(* CoDeSys 2.3.9.59 project: wago_880.pro *)
(* Libraries: WagoLibMBX_01.lib 23.7.19 10:23:10, DALI_647_02_v2.3.lib 13.9.26 18:52:45, DALI_02_v2.14.lib 13.9.26 18:52:45, WagoLibReset.lib 2.12.10 14:48:32, DMXStageProfi_01.lib 13.9.26 18:52:45, SysLibFile.lib 2.12.10 14:48:34, Visual.lib 2.12.10 14:48:34, WagoLibEthernet_01.lib 10.7.18 07:47:36, SysLibSockets.lib 10.2.11 09:20:54, mod_com.lib 2.12.10 14:48:32, KNX_Standard.lib 13.9.26 18:52:45, KNX_IP_750_849_01.lib 13.9.26 18:52:45, Ethernet.lib 2.12.10 14:48:32, SysLibGetAddress.lib 2.12.10 14:48:32, WAGOLibKNXDevice.lib 1.4.16 09:47:39, DALI_647_SensorType2_02.lib 13.9.26 18:52:45, DALI_647_SensorType1_02.lib 13.9.26 18:52:45, Standard.lib 2.12.10 14:48:34, SYSLIBCALLBACK.LIB 2.12.10 14:48:32 *)

(* PLC configuration (modules and I/O channels)
K-Bus [K_Bus] node 0, in %IB0 out %QB0
Fieldbus variables [FB_VARS] node 1, in %IB512 out %QB512
*)

(* Global variable list: Variables_Globales *)
VAR_GLOBAL CONSTANT
	MaxDaliSensors: BYTE := 128;
END_VAR
VAR_GLOBAL
	ConfigDone: BOOL := FALSE; (* Do the config only one time *)
	info : ARRAY[0..63] OF MODULE_INFO; (* I/O Module infos *)

	LedMode: BYTE := 0;

	(* modules infos *)
	nb_module: BYTE;
	nb_module_in: BYTE;
	nb_module_out: BYTE;
	nb_module_analog_in: BYTE;
	nb_module_analog_out: BYTE;
	start_addr_in: WORD;
	start_addr_out: WORD;
	nb_input_digital: WORD;
	nb_output_digital: WORD;

	(* All inputs events *)
	event: ARRAY[0..512] OF INTER_EVENT; (* See Rules mapping below *)
	lights: ARRAY[0..63] OF BYTE;	(* MAX of 256/8 = 32 digital output modules as lights *)
									(* We store only the boolean state of each light *)
	volets: ARRAY[0..512] OF VOLET; (* MAX of 256/8 = 32 digital output modules as volets *)

	HEARTBEAT: BOOL := FALSE;

	OutArrState: ARRAY[0..512] OF BYTE;	(* state of outputs *)

	impulse_time: TIME := T#300ms;

	(* DALI *)
	DALIJoblist: FbDALI_Joblist;

	Dali_switch: DaliSwitch;
	DALIDimmValue: DaliDimValue;
	DALIShowShortAdr: FbDALI_ShowShortAdr;

	(* DALI 647 module *)
	DaliSendValue647: ARRAY[1..64] OF FbDaliSendDimmValue;
	DaliSendValueGrp647: ARRAY[1..16] OF FbDaliSendDimmValue;
	DaliValue647: ARRAY[1..64] OF BYTE;
	DaliValueGrp647: ARRAY[1..16] OF BYTE;

	daliSensors: ARRAY [1..MaxDaliSensors] OF typDaliSensorData;
	DaliSensorT1: ARRAY[1..MaxDaliSensors] OF FbMultiSensorType1;
	DaliButtonT1: ARRAY[1..MaxDaliSensors] OF FbPushbuttonSensorType1;
	DaliSensorT2: ARRAY[1..MaxDaliSensors] OF FbMultiSensorType2;
	DaliButtonT2: ARRAY[1..MaxDaliSensors] OF FbPushbuttonSensorType2;

	(* DALI sensors input mapping *)
	DaliSensorsInputs: ARRAY[0..768] OF BOOL;

	(*
		Modbus addresses mapping:
			- [4096..4352] : Standard digital outputs
			- [6144..6248] : KNX inputs/outputs
			- [6656..7424] : Dali Master Sensors Digital (max 768 addresses available)
			- [256..272] : Dali Master Sensors Analog values (16 addresses for lightlevels in WORD)
	*)

	netOutStandard AT %IB512: ARRAY[0..31] OF BYTE;

	netDaliSensor AT %QB832: ARRAY[0..31] OF BYTE; (* addresses for digital values *)
	netDaliLevels AT %QW256: ARRAY[0..15] OF WORD; (* addresses for light levels *)

	write_word: WRITE_OUTPUT_WORD;
	read_word: READ_INPUT_WORD;
	write_bit: WRITE_OUTPUT_BIT;
	read_bit: READ_INPUT_BIT;

END_VAR
VAR_GLOBAL RETAIN
	(* Rules mapping:
		- [0..256] : standard digital inputs
		- [257..357]: knx digital inputs
	*)
	output_type: ARRAY[0..512] OF OUTPUT_TYPE; (* The type of each output *)
	output_addr: ARRAY[0..512] OF OUTPUT_ADDR; (* The addresses for each type *)

   	volets_position: ARRAY[0..100] OF DWORD;

	(* DMX Values *)
	abDMX_Values: ARRAY [1..255] OF BYTE;
END_VAR

(* Data type *)
TYPE enumDaliSensor :
(
	NoSensor := 0, (* default type is no sensor *)
	MultiSensorType1,
	PushbuttonSensorType1,
	MultiSensorType2,
	PushbuttonSensorType2,
	DaliEcg,
	DaliGroup
);
END_TYPE

(* Data type *)
TYPE OUTPUT_ADDR :
STRUCT

	(* the first ouput address, only needed *)
	ADDR1: BYTE;
	(* the second address used only for the VOLET function bloc *)
	ADDR2: BYTE;

	(* If SameAs <> -1, then a input is wired the same as the specified ID *)
	SameAs: INT := -1;

END_STRUCT
END_TYPE

(* Data type *)
(* Enumerate all type of output.
	NONE: Do nothing.
	TELERUPTEUR: Simulate a telerupteur.
	DIRECT: The input is directly "wired" to the output.
	VOLET: Simulate a volet with one button and 2 output (up and down).
	TELERUPTEUR_DALI: Controls a DALI lamp
	TELERUPTEUR_DALI_GROUP: Controls a DALI group
	KNX_OUTPUT: Simulate a telerupteur with a KNX bool output
*)

TYPE OUTPUT_TYPE : (NONE,
					TELERUPTEUR, DIRECT,
					VOLET, VOLET_IMPULSE,
					TELERUPTEUR_DALI,
					TELERUPTEUR_DALI_GROUP,
					TELERUPTEUR_KNX_OUTPUT,
					DIRECT_KNX_OUTPUT);
END_TYPE

(* Data type *)
TYPE typDaliSensorData :
STRUCT

	SensorType: enumDaliSensor;

	(* MultiSensorType1 *)
	AddrPresence: BYTE;
	AddrLightLevel: BYTE;
	offDelay: TIME;

	(* MultiSensorType2 *)
	AddrRemote: BYTE;

	(* PushbuttonSensorType1 *)
	AddrButton1: BYTE;
	AddrButton2: BYTE;
	AddrButton3: BYTE;
	AddrButton4: BYTE;

	(* PushbuttonSensorType2 *)
	AddrButtons: BYTE;

	(* Dali devices *)
	Address: BYTE;

END_STRUCT
END_TYPE

(* Data type *)
TYPE typEthernet_BUFFER :
	STRUCT
		Index		:	INT;
		Data		:	ARRAY[1..1500] OF BYTE;
	END_STRUCT
END_TYPE

(* Data type *)
(* Enumerate all type of output.
	NONE: Do nothing.
	TELERUPTEUR: Simulate a telerupteur.
	DIRECT: The input is directly "wired" to the output.
	VOLET: Simulate a volet with one button and 2 output (up and down).
*)

TYPE VOLET_MODE : (VOLET_STOP, VOLET_UP, VOLET_DOWN, IMP_UP, IMP_DOWN, IMP_STOP);
END_TYPE

(* POU PLC_PRG, ST *)
PROGRAM PLC_PRG
VAR
	i: INT;
	j: INT;
	start: BYTE;
	init_dali: BOOL := FALSE;
	valw: WORD;

	led: LedUsr;

END_VAR
(* Main PRG *)
Config_File_XML();

(*DaliReadCsvFile(xStart := TRUE);*)

led(Mode := LedMode);

(* Start the config program *)
Config;

IF (Config.CONFIG_DALI = TRUE) THEN
	(* Call DALI jobs to send commands on the DALI bus *)
	DALIJoblist();
	DALI_Config();
END_IF

(* Read inputs and send their status on the network if they changed *)
SendInput;

(* Read a command from UDP *)
UDPServer;

IF (HEARTBEAT = FALSE) THEN
 	ManageOutput;
END_IF

(* Run the DALI FB for 647 module *)
IF Config.CONFIG_DALI_647 = TRUE THEN
	DaliPrg647;
END_IF

IF (HEARTBEAT = FALSE) THEN

	j := start_addr_out / 8;
	FOR i := start_addr_out / 16 TO 255 DO
		valw := OutArrState[j + 1];
		write_word(WORD_ADDRESS := i, VALUE := SHL(valw, 8) + OutArrState[j]);
		j := j + 2;
	END_FOR
ELSE

	j := 0;
	FOR i := 0 TO 14 DO
		valw := netOutStandard[j + 1];
		write_word(WORD_ADDRESS := i + start_addr_out / 16, VALUE := SHL(valw, 8) + netOutStandard[j]);
		j := j + 2;
		OutArrState[j] := netOutStandard[j];
		OutArrState[j + 1] := netOutStandard[j + 1];
	END_FOR

END_IF
END_PROGRAM

(* POU LedUsr, ST *)
FUNCTION_BLOCK LedUsr
VAR_INPUT
	Mode: BYTE;

END_VAR
VAR_OUTPUT
END_VAR
VAR
	Sequence: ARRAY [0..4] OF FLASHING_SEQUENCE;
	ptrFS: POINTER TO FLASHING_SEQUENCE;

	i: BYTE := 0;
END_VAR
CASE Mode OF
	0 : i := 0;
	1 : i := 11; (* Mode Wago *)
	2 : i := 12; (* Mode PC *)
	3 : i := 13; (* Error *)
END_CASE

LedMode := 255;

CASE i OF
	0 : (* Init *)
		Sequence[0].Colour := ORANGE;
		Sequence[0].Frequency := 10;
		Sequence[0].Relation := 128;
		Sequence[0].Duration := t#0s;

		Sequence[1].Colour := ORANGE;
		Sequence[1].Frequency := 0;
		Sequence[1].Relation := 128;
		Sequence[1].Duration := t#0s;

		Sequence[2].Colour := GREEN;
		Sequence[2].Frequency := 0;
		Sequence[2].Relation := 128;
		Sequence[2].Duration := t#0s;

		Sequence[3].Colour := RED;
		Sequence[3].Frequency := 0;
		Sequence[3].Relation := 128;
		Sequence[3].Duration := t#0s;

		Sequence[4].Colour := ORANGE;
		Sequence[4].Frequency := 0;
		Sequence[4].Relation := 0;
		Sequence[4].Duration := t#0s;

		ptrFS := ADR(Sequence);
		SET_FLASHING_SEQUENCE(TRUE, ADR(ptrFS));

		i := 10;

	10: (* Start *)
		SET_FLASHING_SEQUENCE_INDEX(TRUE, TRUE, 0);
		START_FLASHING_SEQUENCE(TRUE);

		i := 255;

	11: (* Led Mode wago *)
		SET_FLASHING_SEQUENCE_INDEX(TRUE, TRUE, 1);

		i := 255;

	12: (* Led Mode PC *)
		SET_FLASHING_SEQUENCE_INDEX(TRUE, TRUE, 2);

		i := 255;

	13: (* Led Error *)
		SET_FLASHING_SEQUENCE_INDEX(TRUE, TRUE, 3);

		i := 255;

END_CASE
END_FUNCTION_BLOCK

(* POU Config_File_XML, ST *)
PROGRAM Config_File_XML
VAR RETAIN
	wModuleCount : WORD;
END_VAR
VAR CONSTANT
	STRING_1: STRING := '<?xml version="1.0" encoding="ISO-8859-1"?>$r$n';
	STRING_2: STRING := '<?xml-stylesheet type="text/xsl" href="/webserv/cplcfg/EA-config.xsl" ?>$R$n';
	STRING_3: STRING := '<WAGO>$R$n';
	STRING_4: STRING := '<Module ARTIKELNR="" MAP="PLC" LOC="ALL"></Module>$R$n';
	STRING_5: STRING := '</WAGO>$r$n';
END_VAR
VAR
	info : ARRAY[0..63] OF MODULE_INFO;
	access: MODULE_INFO_ACCESS;
	i: INT := 0;
	Status: BYTE := 0;
	DetectedModules: INT;
	FileHandle: DWORD;
	dwWrite: DWORD;
	NumberOfEntries: BYTE := 0;
	FileIsClosed: BOOL;
END_VAR
CASE Status OF
	0 :	ADD_PI_INFORMATION(EN:=TRUE, pAccess:=ADR(access), pInfo:=ADR(info));
		i:=0;
		WHILE info[i].physicalPos<>0
			DO
			i:=i+1;
		END_WHILE
		DetectedModules := i;
		Status := Status +1;
	1 :	IF DetectedModules = wModuleCount
			THEN
			Status := 255; (* Done *)
		ELSE
			Status := 10;
		END_IF
	10:	FileHandle:=SysFileOpen(FileName:='\etc\EA-config.xml', Mode:='w');
		IF FileHandle <> 0 THEN
			Status := Status+1;
		END_IF
	11:	dwWrite:=SysFileWrite(File:=FileHandle, Buffer:=ADR(STRING_1), Size:=LEN(STRING_1));
		IF dwWrite=LEN(STRING_1) THEN
			Status := Status+1;
		END_IF
	12:	dwWrite:=SysFileWrite(File:=FileHandle, Buffer:=ADR(STRING_2), Size:=LEN(STRING_2));
		IF dwWrite=LEN(STRING_2) THEN
			Status := Status+1;
		END_IF
	13:	dwWrite:=SysFileWrite(File:=FileHandle, Buffer:=ADR(STRING_3), Size:=LEN(STRING_3));
		IF dwWrite=LEN(STRING_3) THEN
			Status := Status+1;
		END_IF
	14:	dwWrite:=SysFileWrite(File:=FileHandle, Buffer:=ADR(STRING_4), Size:=LEN(STRING_4));
		IF dwWrite=LEN(STRING_4) THEN
			Status := Status+1;
			NumberOfEntries := NumberOfEntries+1;
		END_IF
	15: IF NumberOfEntries < DetectedModules
			THEN
			Status := Status -1;
		ELSE
			Status := Status +1;
		END_IF
	16:	dwWrite:=SysFileWrite(File:=FileHandle, Buffer:=ADR(STRING_5), Size:=LEN(STRING_5));
		IF dwWrite=LEN(STRING_5) THEN
			Status := Status+1;
		END_IF
	17:	FileIsClosed := SysFileClose(File:= FileHandle);
		IF FileIsClosed
			THEN
			Status := 20;
		END_IF
	20:	wModuleCount := DetectedModules;
		FirmwareReset(EN := TRUE);
END_CASE
END_PROGRAM

(* POU Config, ST *)
PROGRAM Config
VAR
	access : MODULE_INFO_ACCESS;
	cpt: BYTE;
	ethernet_config : ETHERNET_SET_VARIABLES;
	CONFIG_DALI: BOOL := FALSE;
	CONFIG_DALI_647: BOOL := FALSE;
	first_in: BOOL := FALSE;
	first_out: BOOL := FALSE;
	AddrDali647In: INT;
	AddrDali647Out: INT;
END_VAR
VAR_INPUT RETAIN
	SERVER_IP: DWORD;
	DALI_MODE: BYTE;
END_VAR
VAR CONSTANT
	CALAOS_VERSION_H: WORD := 3;
	CALAOS_VERSION_L: WORD := 0;
	DALI: BYTE := 1;
	DSI: BYTE := 2;
END_VAR
(* Do all the config job *)

IF (ConfigDone = FALSE) THEN

(* Get the module I/O Config *)
access.physicalPosTo := 0;
access.moduleType := 0;
ADD_PI_INFORMATION( 1, ADR(access), ADR(info[0]) );

FOR cpt := 0 TO 63 DO
	IF (info[cpt].moduleType = 0 AND info[cpt].physicalPos = 0) THEN
		cpt := 63; (* the end *)
	ELSE
		IF (info[cpt].moduleType = 641) THEN
			(* This is a DALI 641 module *)
			CONFIG_DALI := TRUE;
		END_IF

		IF (info[cpt].moduleType = 647) THEN
			(* This is a DALI 753-647 module (multi master) *)
			CONFIG_DALI_647 := TRUE;
		END_IF

		nb_module := nb_module + 1;
		IF ((info[cpt].desc.sizePAE > 8) AND (info[cpt].desc.channels > 0)) THEN
			nb_module_analog_in := nb_module_analog_in + 1;
(*			start_addr_in := start_addr_in + info[cpt].desc.sizePAE; *)
			IF CONFIG_DALI_647 = FALSE THEN
				AddrDali647In := AddrDali647In + (info[cpt].desc.sizePAE / 8);
			END_IF
		END_IF
		IF ((info[cpt].desc.sizePAA > 8) AND (info[cpt].desc.channels > 0)) THEN
			nb_module_analog_out := nb_module_analog_out + 1;
(*			start_addr_out := start_addr_out + info[cpt].desc.sizePAA; *)
			IF CONFIG_DALI_647 = FALSE THEN
				AddrDali647Out := AddrDali647Out + (info[cpt].desc.sizePAA / 8);
			END_IF
		END_IF
		IF ((info[cpt].desc.sizePAE <= 16) AND (info[cpt].desc.sizePAE > 0) AND (info[cpt].desc.channels = 0)) THEN
			nb_module_in := nb_module_in + 1;
			nb_input_digital := nb_input_digital + info[cpt].desc.sizePAE;

			IF (first_in = FALSE) THEN
				first_in := TRUE;
				start_addr_in := info[cpt].desc.posPAE;
			END_IF
		END_IF
		IF ((info[cpt].desc.sizePAA <= 16) AND (info[cpt].desc.sizePAA > 0) AND (info[cpt].desc.channels = 0)) THEN
			nb_module_out := nb_module_out + 1;
			nb_output_digital := nb_output_digital + info[cpt].desc.sizePAA;

			IF (first_out = FALSE) THEN
				first_out := TRUE;
				start_addr_out := info[cpt].desc.posPAA;
			END_IF
		END_IF

	END_IF
END_FOR

(* Start the heartbeat timer *)
(*HEARTBEAT_TIMER(IN:=FALSE, PT:=T#30s);*)
(*HEARTBEAT_TIMER(IN:=TRUE, PT:=T#30s);*)

(* Config du timout des sockets *)
ethernet_config(EN:=TRUE, BootpRequest:=0, ConnectionWdTime:=65535);

ConfigDone := TRUE;

END_IF
END_PROGRAM

(* POU SendInput, ST *)
PROGRAM SendInput
VAR
	cpt: INT;

	eth: Ethernet_Client;
	wBuffer: POINTER TO BYTE;
	command: STRING(255);
	start_send: BOOL := FALSE;
	ReceiveData: typEthernet_buffer;
	Write: ETHERNET_WRITE_PT;
	socket:	WORD;
END_VAR
(* Get all inputs *)

(* Get the address of the first digital input *)
FOR cpt := 0 TO UINT_TO_BYTE(nb_input_digital) - 1 DO
	event[cpt](IN := GetInput(cpt + start_addr_in));

	(* Send inputs to network *)
	IF (event[cpt].ON = TRUE) THEN
		command := 'WAGO INT ';
		command := CONCAT(command,  INT_TO_STRING(cpt));
		command := CONCAT(command,  ' 1');

		Write(EN := 0, SOCKET := 0, LEN_IN := 0, DST_IP:=0, DST_PORT:=0, DATA_PT := wBuffer);
		Write(EN := 1, SOCKET := socket, LEN_IN := LEN(command), DST_IP := Config.SERVER_IP, DST_PORT := 4646, DATA_PT := wBuffer);
	END_IF
	IF (event[cpt].OFF = TRUE) THEN
		command := 'WAGO INT ';
		command := CONCAT(command,  INT_TO_STRING(cpt));
		command := CONCAT(command,  ' 0');

		Write(EN := 0, SOCKET := 0, LEN_IN := 0, DST_IP:=0, DST_PORT:=0, DATA_PT := wBuffer);
		Write(EN := 1, SOCKET := socket, LEN_IN := LEN(command), DST_IP := Config.SERVER_IP, DST_PORT := 4646, DATA_PT := wBuffer);
	END_IF
END_FOR

wBuffer := ADR(command);

eth(xOPEN_CLIENT := TRUE, wIP := Config.SERVER_IP, wPort := 4646,
	xTCP_PROTOCOL := FALSE, iBYTES_TO_SEND := LEN(command) + 1,
	ptSEND_BUFFER := wBuffer, xSTART_SEND := start_send,
	utRECEIVE_BUFFER := ReceiveData);

socket := eth.MyEthernetOpen.SOCKET;
END_PROGRAM

(* POU Ethernet_Client, ST *)
FUNCTION_BLOCK Ethernet_Client
(************************************************************)
(* ETHERNET_CLIENT		                             			*)
(* Ver. 1.0                                      			          			*)
(* Date    :  10.02.2003					          			*)
(* Author :  Volker Begemann                                       		*)
(************************************************************)
VAR_INPUT
	xOPEN_CLIENT			:	BOOL;			(* Set TRUE to enable function block			*)
	wIP						:	DWORD;		(* IP Address of server						*)
	wPORT					:	WORD;		(* Port number								*)
	xTCP_PROTOCOL		:	BOOL;			(* TRUE => TCP; FALSE => UDP				*)
	iBYTES_TO_SEND		:	INT;			(* Number of bytes to transmit				*)
	ptSEND_BUFFER			:	POINTER TO ARRAY[1..1500] OF BYTE;	(* Transmit Buffer	*)
END_VAR
VAR_IN_OUT
	xSTART_SEND			:	BOOL;			(* Set TRUE to initiate data transmittal, will be	*)
													(* reset FALSE when transmittal is completed 	*)
	utRECEIVE_BUFFER		:	typEthernet_BUFFER;	(* Receive Buffer *)
END_VAR
VAR_OUTPUT
	utERROR					:	ETH_ERROR;	(* See ETH_ERROR datatype in ETHERNET.LIB	*)
													(* for error codes and definitions						*)
	xCLIENT_OPEN			:	BOOL;			(* TRUE if socket connection made					*)
	wSOCKET					:	WORD;		(* Socket connection number							*)
END_VAR
VAR
	MyEthernetOpen				: ETHERNET_CLIENT_OPEN;
	MyEthernetClose				: ETHERNET_CLIENT_CLOSE;
	MyEthernetWrite				: ETHERNET_WRITE;
	MyEthernetRead				: ETHERNET_READ;
	EthernetBuffer					: ARRAY[1..1500] OF BYTE;
	Status							: WORD:=0;
	i								: INT;
	GetConfig						: ETHERNET_GET_NETWORK_CONFIG;
	Protocol						: WORD;
	ProtocolType					: WORD;
	CloseState						:INT;
END_VAR
IF xOpen_Client THEN

	CASE Status OF
		0:(*Initialize functionblocks*)
			GetConfig(EN:=FALSE );
			GetConfig(EN:=TRUE );
			status:=1;
			utERROR:=0;
			wSocket:=0;
			closeState:=0;
			xCLIENT_OPEN:=FALSE;

			IF xTCP_PROTOCOL THEN
				Protocol		:= IPPROTO_TCP; (*TCP*)
				ProtocolType	:= SOCK_STREAM;
			ELSE
				Protocol		:= IPPROTO_UDP;(*UDP*)
				ProtocolType	:= SOCK_DGRAM;
			END_IF

		1:(*check ethernet stack*)
			GetConfig(EN:=TRUE );
			IF GetConfig.ENO THEN
				IF GetConfig.IP_ADR<>0 THEN
					status:=4;(*stack initialized*)
				ELSE
					status:=0;(*try again*)
				END_IF
			END_IF

	
		4:(*open connection*)
			MyEthernetRead(	EN:= 0, SOCKET:=0 ,  DATA:=EthernetBuffer );
			MyEthernetClose(EN:= 0);
			MyEthernetOpen(EN:=0);

			MyEthernetOpen(EN:=1 , TYP:=ProtocolType	 , PROTO:=Protocol , IP_ADR:= wIP, PORT:=wPort );

			status:=5;

		5:(*wait for server response according to client  request to open the connection*)
			MyEthernetOpen(EN:=1, TYP:=ProtocolType, PROTO:=Protocol, IP_ADR:= wIP, PORT:=wPort );
			IF  MyEthernetOpen.ENO = 1 THEN
				IF MyEthernetOpen.ERROR = 0 THEN
					Status  := 10; (*socket available*)
					xCLIENT_OPEN:=TRUE;
					wSOCKET	:=MyEthernetOpen.socket;
				ELSE
					Status := 0; (*no socket available, try it again *)
				END_IF;
				utERROR:=MyEthernetOpen.ERROR;
			END_IF


		10:(* Monitor ethernet port for new data *)

	 		MyEthernetRead(	EN:= 1, SOCKET:=MyEthernetOpen.SOCKET ,  DATA:=EthernetBuffer );
			MyEthernetRead(	EN:= 0, SOCKET:=0 ,  DATA:=EthernetBuffer );

			utERROR:=MyEthernetREAD.ERROR;
			IF(MyEthernetRead.ERROR<>0) THEN  (* Error reading the socket, close it *)
				Status:=40;
			ELSIF (MyEthernetRead.LEN_OUT <>0) THEN  (* Process the data received via the ethernet port *)
				Status:=20;
				ELSIF (iBytes_TO_SEND > 0 AND xSTART_SEND) THEN  (* Process the data put in the send_buffer *)
				status:=30;
				MyEthernetWrite(	EN:= 0 , DATA:=EthernetBuffer );
			END_IF

		20:	(* Copy the data received via the ethernet port to the receive buffer*)

			FOR i := 1 TO MyEthernetRead.LEN_OUT DO
				utReceive_buffer.index :=(utReceive_buffer.index MOD 1500)+1;
				utReceive_buffer.data[utReceive_buffer.index] := EthernetBuffer[i];
			END_FOR
			Status:=10;

		30: (* Process the data in the send buffer *)

			EthernetBuffer :=ptSEND_BUFFER^;
			MyEthernetWrite(	EN:= 1,SOCKET:= MyEthernetOpen.SOCKET,
								LEN_IN:=iBYTES_TO_SEND,DATA:=EthernetBuffer );

			IF MyEthernetWrite.eno THEN
				IF(MyEthernetWrite.ERROR <>0) THEN
					Status:=40;(* Error writing to the socket, close it *)
				ELSE
					Status:=10; (* Comms complete, read more data *)
				END_IF;
				xSTART_SEND:=FALSE;
				utERROR:=MyEthernetWrite.ERROR;
			END_IF

		40:	(* Close the client *)

			MyEthernetClose(EN:= 1, SOCKET:= MyEthernetOpen.SOCKET);
			IF MyEthernetClose.eno THEN
				MyEthernetClose(EN:= 0);
				xCLIENT_OPEN:=FALSE;
				Status := 0; (* Try to open the server again *)
			END_IF
	
	END_CASE;
ELSE
	CASE CloseState OF
	0:
		MyEthernetClose(EN:= 0);
		MyEthernetClose(EN:= 1, SOCKET:= MyEthernetOpen.SOCKET);
		CloseState:=1;
	1:
		MyEthernetClose(EN:= 1, SOCKET:= MyEthernetOpen.SOCKET);
		IF MyEthernetClose.eno THEN
			MyEthernetClose(EN:= 0);
			CloseState:=2;
		END_IF
	2:
		Status := 0;
		utERROR:=0;
		xCLIENT_OPEN:=FALSE;
	END_CASE
END_IF
END_FUNCTION_BLOCK

(* POU GetInput, ST *)
FUNCTION GetInput : BOOL
VAR_INPUT
	bit_offset: UINT;
END_VAR
VAR
END_VAR
VAR CONSTANT
	byBitArr: ARRAY[0..7] OF BYTE := 16#01,16#02,16#04,16#08,16#10,16#20,16#40,16#80;
END_VAR
(* get the byte AND  select the bit *)

read_bit(WORD_ADDRESS := bit_offset / 16, BIT_ADDRESS := bit_offset MOD 16);

GetInput := read_bit.VALUE;
END_FUNCTION

(* POU UDPServer, ST *)
PROGRAM UDPServer
VAR
	server: EthernetServer_FB;

	rBuffer, wBuffer: POINTER TO BYTE;
	buffer: ARRAY[1 .. 1500] OF BYTE;
	cmd: STRING(255);
	start_send: BOOL := FALSE;
	i: WORD;
	dali_group: BOOL;

	HEARTBEAT_TIMER: TON;

	p1: DINT;
	p2: DINT;
	p3: DINT;
	p4: DINT;
	p5: DINT;
	p6: DINT;
	p7: DINT;
	p8: DINT;
	ip1, ip2, ip3, ip4: DWORD;
	DaliSend: BOOL := FALSE;

	(* Used by dali config for answer
	   0 = no action
	   1 = Search all active address
	   2 = Read groups for short adress
	   3 = Switch on/off all lamps
	  98 = Addresing query
	  99 = Addressing in progress
	*)
	DaliSendAction: BYTE := 0;

	(* Dali config FB *)
	DALIShowShortAdr: FbDALI_ShowShortAdr;
	DALIConfigDevice: FbDALI_ConfigDevice;
	DALIConfigShortAddress: FbDALI_ConfigShortAddress;
	DALIMaster: FbDALI_Master;
	DALIMasterAdv: FbDALI_Master_Adv;

	extendedAddr: BOOL;
	newAddressing: BOOL;
	resetAddr: BOOL;
	replaceAddr: BOOL;
	delAddressing: BOOL;
	oldAddr, newAddr, delAddr: BYTE;
	dali_master: BOOL;
	group_address: BYTE;
	groups_cmd_1_8: BYTE;
	addr_1_16: WORD;
	addr_17_32: WORD;

	dmx_read_addr: BYTE;

	daliShortAddr: BYTE;

END_VAR
(* Here we start an UDP server for other network functions *)

HEARTBEAT_TIMER(IN:=TRUE, PT:=T#30s);

rBuffer := ADR(buffer);
wBuffer := ADR(cmd);

(* cmd := CONCAT(cmd, ASCIIBYTE_TO_STRING(0)); *)

server.tTIMEOUT	:= t#60s;
server.xTCP_PROTOCOL := FALSE;
server.wPORT := 4646;
server.iBYTES_TO_SEND := LEN(cmd) + 1;
server(xOPEN_SERVER := TRUE, xSTART_SEND := start_send, ptSEND_BUFFER := wBuffer, ptRECV_BUFFER := rBuffer);

IF server.bDataReceived THEN

	cmd := '';
	FOR i := 1 TO server.iBYTES_RECEIVED DO
		cmd := CONCAT(cmd, ASCIIBYTE_TO_STRING(buffer[i]));
	END_FOR

	IF (STRING_COMPARE(cmd, 'WAGO_HEARTBEAT') = TRUE) THEN
		HEARTBEAT_TIMER(IN:=FALSE, PT:=T#30s);
		HEARTBEAT_TIMER(IN:=TRUE, PT:=T#30s);

		LedMode := 2;
	END_IF

	IF (Strncmp(cmd, 'WAGO_SET_OUTTYPE ', 17) = TRUE) THEN
		p1 := GET_PARAM_DINT(cmd, 1);
		p2 := GET_PARAM_DINT(cmd, 2);
		CASE p2 OF
		0: output_type[p1] := NONE;
		1: output_type[p1] := TELERUPTEUR;
		2: output_type[p1] := DIRECT;
		3: output_type[p1] := VOLET;
		4: output_type[p1] := VOLET_IMPULSE;
		5: output_type[p1] := TELERUPTEUR_DALI;
		6: output_type[p1] := TELERUPTEUR_DALI_GROUP;
		7: output_type[p1] := TELERUPTEUR_KNX_OUTPUT;
		8: output_type[p1] := DIRECT_KNX_OUTPUT;
		END_CASE
	END_IF

	IF (Strncmp(cmd, 'WAGO_SET_OUTADDR ', 17) = TRUE) THEN
		p1 := GET_PARAM_DINT(cmd, 1);
		p2 := GET_PARAM_DINT(cmd, 2);
		p3 := GET_PARAM_DINT(cmd, 3);
		p4 := GET_PARAM_DINT(cmd, 4);
		output_addr[p1].ADDR1 := DINT_TO_BYTE(p2);
		output_addr[p1].ADDR2 := DINT_TO_BYTE(p3);
		output_addr[p1].SameAs := DINT_TO_INT(p4);
	END_IF

	IF (Strncmp(cmd, 'WAGO_GET_OUTTYPE ', 17) = TRUE) THEN
		p1 := GET_PARAM_DINT(cmd, 1);
		cmd := 'WAGO_OUTTYPE ';
		cmd := CONCAT(cmd, ITOA(DINT_TO_INT(p1)));
		cmd := CONCAT(cmd, ' ');
		CASE output_type[p1] OF
		NONE: cmd := CONCAT(cmd, ITOA(0));;
		TELERUPTEUR: cmd := CONCAT(cmd, ITOA(1));;
		DIRECT: cmd := CONCAT(cmd, ITOA(2));;
		VOLET: cmd := CONCAT(cmd, ITOA(3));;
		VOLET_IMPULSE: cmd := CONCAT(cmd, ITOA(4));;
		TELERUPTEUR_DALI: cmd := CONCAT(cmd, ITOA(5));;
		TELERUPTEUR_DALI_GROUP: cmd := CONCAT(cmd, ITOA(6));;
		TELERUPTEUR_KNX_OUTPUT: cmd := CONCAT(cmd, ITOA(7));;
		DIRECT_KNX_OUTPUT: cmd := CONCAT(cmd, ITOA(8));;
		END_CASE
		start_send := TRUE;
	END_IF

	IF (Strncmp(cmd, 'WAGO_GET_OUTADDR ', 17) = TRUE) THEN
		p1 := GET_PARAM_DINT(cmd, 1);
		cmd := 'WAGO_OUTADDR ';
		cmd := CONCAT(cmd, ITOA(DINT_TO_INT(p1)));
		cmd := CONCAT(cmd, ' ');
		cmd := CONCAT(cmd, ITOA(output_addr[p1].ADDR1));
		cmd := CONCAT(cmd, ' ');
		cmd := CONCAT(cmd, ITOA(output_addr[p1].ADDR2));
		cmd := CONCAT(cmd, ' ');
		cmd := CONCAT(cmd, ITOA(output_addr[p1].SameAs));
		start_send := TRUE;
	END_IF

	IF (STRING_COMPARE(cmd, 'WAGO_GET_INFO') = TRUE) THEN
		cmd := 'WAGO_INFO ';
		cmd := CONCAT(cmd, ITOA(nb_module));
		cmd := CONCAT(cmd, ' ');
		cmd := CONCAT(cmd, ITOA(nb_module_in));
		cmd := CONCAT(cmd, ' ');
		cmd := CONCAT(cmd, ITOA(WORD_TO_INT(nb_module_out)));
		cmd := CONCAT(cmd, ' ');
		cmd := CONCAT(cmd, ITOA(WORD_TO_INT(nb_input_digital)));
		cmd := CONCAT(cmd, ' ');
		cmd := CONCAT(cmd, ITOA(WORD_TO_INT(nb_output_digital)));
		cmd := CONCAT(cmd, ' ');
		cmd := CONCAT(cmd, ITOA(nb_module_analog_in));
		cmd := CONCAT(cmd, ' ');
		cmd := CONCAT(cmd, ITOA(nb_module_analog_out));
		start_send := TRUE;
	END_IF

	IF (Strncmp(cmd, 'WAGO_GET_INFO_MODULE ', 21) = TRUE) THEN
		p1 := GET_PARAM_DINT(cmd, 1);
		cmd := 'WAGO_MODULE ';
		cmd := CONCAT(cmd, ITOA(DINT_TO_INT(p1)));
		cmd := CONCAT(cmd, ' ');
		cmd := CONCAT(cmd, ITOA(WORD_TO_INT(info[p1].moduleType)));
		cmd := CONCAT(cmd, ' ');
		cmd := CONCAT(cmd, ITOA(info[p1].physicalPos));
		cmd := CONCAT(cmd, ' ');
		cmd := CONCAT(cmd, ITOA(info[p1].desc.sizePAE));
		cmd := CONCAT(cmd, ' ');
		cmd := CONCAT(cmd, ITOA(info[p1].desc.sizePAA));
		start_send := TRUE;
	END_IF

	IF (Strncmp(cmd, 'WAGO_SET_SERVER_IP ', 19) = TRUE) THEN
		cmd := DELETE(cmd, 19, 1);
		(* deletes the dot  *)
		cmd := REPLACE(cmd, ' ', 1, FIND(cmd, '.'));
		cmd := REPLACE(cmd, ' ', 1, FIND(cmd, '.'));
		cmd := REPLACE(cmd, ' ', 1, FIND(cmd, '.'));
		ip1 := GET_PARAM_DINT(cmd, 0);
		ip2 := GET_PARAM_DINT(cmd, 1);
		ip3 := GET_PARAM_DINT(cmd, 2);
		ip4 := GET_PARAM_DINT(cmd, 3);
		Config.SERVER_IP := SHL(ip1, 24) OR SHL(ip2, 16) OR SHL(ip3, 8) OR ip4;
	END_IF


	IF (Strncmp(cmd, 'WAGO_SET_DMX_IP ', 16) = TRUE) THEN
		cmd := DELETE(cmd, 16, 1);
		DMX.IPaddress := cmd;
	END_IF

	IF (Strncmp(cmd, 'WAGO_SET_OUTPUT ', 16) = TRUE) THEN
		p1 := GET_PARAM_DINT(cmd, 1);
		p2 := GET_PARAM_DINT(cmd, 2);

		p1 := start_addr_out + p1;

		IF (p2 = 1) THEN
			SetOutput(DINT_TO_UINT(p1), TRUE);
		ELSE
			SetOutput(DINT_TO_UINT(p1), FALSE);
		END_IF
	END_IF

	IF (Strncmp(cmd, 'WAGO_GET_VERSION', 16) = TRUE) THEN
		cmd := 'WAGO_GET_VERSION ';
		cmd := CONCAT(cmd, ITOA(WORD_TO_INT(Config.CALAOS_VERSION_H)));
		cmd := CONCAT(cmd, '.');
		cmd := CONCAT(cmd, ITOA(WORD_TO_INT(Config.CALAOS_VERSION_L)));
		cmd := CONCAT(cmd, ' 750-849');
		start_send := TRUE;
	END_IF

	IF (Strncmp(cmd, 'WAGO_DALI_SET ', 14) = TRUE) THEN
		p1 := GET_PARAM_DINT(cmd, 1); (* Dali Line *)
		p2 := GET_PARAM_DINT(cmd, 2); (* Short addr or group? *)
		p3 := GET_PARAM_DINT(cmd, 3); (* Dali Address *)
		p4 := GET_PARAM_DINT(cmd, 4); (* Dimm value in percent *)
		p5 := GET_PARAM_DINT(cmd, 5); (* Fade time *)

		IF (p2 = 1) THEN
			dali_group := TRUE;
		ELSE
			dali_group := FALSE;
		END_IF

		IF (p3 > 99) THEN
			abDMX_Values[DINT_TO_BYTE(p3 - 100)] := DINT_TO_BYTE(p4 * 255 / 100);
		ELSE
			Dali_switch(bAddress := DINT_TO_BYTE(p3), xGroup := dali_group, xButton := FALSE);
			Dali_switch(bAddress := DINT_TO_BYTE(p3), xGroup := dali_group, bDimmLevel := DINT_TO_BYTE(p4),
				bFadeTime := DINT_TO_BYTE(p5), xButton := TRUE);
		END_IF
	END_IF

	IF (Strncmp(cmd, 'WAGO_DALI_GET ', 14) = TRUE) THEN
		p1 := GET_PARAM_DINT(cmd, 1); (* Dali Line *)
		p2 := GET_PARAM_DINT(cmd, 2); (* Short addr *)
		p3 := GET_PARAM_DINT(cmd, 3); (* Short addr or group? *)

		IF (p3 = 1) THEN
			dali_group := TRUE;
		ELSE
			dali_group := FALSE;
		END_IF

		IF (p2 < 99) THEN
			IF Config.CONFIG_DALI = TRUE THEN
				DALIDimmValue(xEnable := TRUE, bShortAddress := DINT_TO_BYTE(p2), tCycleTime := t#1s);
			END_IF
			daliShortAddr := DINT_TO_BYTE(p2);
			dmx_read_addr := 0;
		ELSE
			dmx_read_addr := DINT_TO_BYTE(p3 - 100);
		END_IF
		DaliSend := TRUE;
	END_IF

    IF (Strncmp(cmd, 'WAGO_INFO_VOLET_GET ', 20) = TRUE) THEN
		p1 := GET_PARAM_DINT(cmd, 1);
		cmd := 'WAGO_INFO_VOLET ';
		cmd := CONCAT(cmd, ITOA(DINT_TO_INT(p1)));
		cmd := CONCAT(cmd, ' ');
		cmd := CONCAT(cmd, DWORD_TO_STRING(volets_position[p1]));
		start_send := TRUE;
	END_IF

    IF (Strncmp(cmd, 'WAGO_INFO_VOLET_SET ', 20) = TRUE) THEN
		p1 := GET_PARAM_DINT(cmd, 1);
		p2 := GET_PARAM_DINT(cmd, 2);
		volets_position[p1] := DINT_TO_DWORD(p2);
	END_IF

		IF (Strncmp(cmd, 'WAGO_DALI_GET_ADDR ', 18) = TRUE) THEN
		p1 := GET_PARAM_DINT(cmd, 1);
		dali_master := TRUE;
		DALIMasterAdv(xStartDaliMaster := dali_master, iCommand := 506);
		DaliSendAction := 1;
	END_IF

	IF (Strncmp(cmd, 'WAGO_DALI_GET_DEVICE_INFO ', 26) = TRUE) THEN
		p1 := GET_PARAM_DINT(cmd, 1);
		p2 := GET_PARAM_DINT(cmd, 2);
		DALIConfigDevice(xQuery := FALSE);
		DALIConfigDevice(xQuery := TRUE, bAddress := DINT_TO_BYTE(p2));
		DaliSendAction := 2;
	END_IF

	IF (Strncmp(cmd, 'WAGO_DALI_GET_DEVICE_GROUP ', 27) = TRUE) THEN
		p1 := GET_PARAM_DINT(cmd, 1);
		p2 := GET_PARAM_DINT(cmd, 2); (* address *)
		group_address := DINT_TO_BYTE(p2);
		dali_master := TRUE;
		DALIMaster(xStartDaliMaster := dali_master, iCommand := 192, bAddress := group_address);
		DaliSendAction := 3;
	END_IF

	IF (Strncmp(cmd, 'WAGO_DALI_DEVICE_ADD_GROUP ', 27) = TRUE) THEN
		p1 := GET_PARAM_DINT(cmd, 1);
		p2 := GET_PARAM_DINT(cmd, 2); (* device address *)
		p3 := GET_PARAM_DINT(cmd, 3); (* group *)
		dali_master := TRUE;
		DALIMasterAdv(xStartDaliMaster := dali_master, iCommand := 501, bCommandValue1 := 95 + DINT_TO_BYTE(p3), bAddress := DINT_TO_BYTE(p2));
		DaliSendAction := 5;
	END_IF

	IF (Strncmp(cmd, 'WAGO_DALI_DEVICE_DEL_GROUP ', 27) = TRUE) THEN
		p1 := GET_PARAM_DINT(cmd, 1);
		p2 := GET_PARAM_DINT(cmd, 2); (* device address *)
		p3 := GET_PARAM_DINT(cmd, 3); (* group *)
		dali_master := TRUE;
		DALIMasterAdv(xStartDaliMaster := dali_master, iCommand := 501, bCommandValue1 := 111 + DINT_TO_BYTE(p3), bAddress := DINT_TO_BYTE(p2));
		DaliSendAction := 6;
	END_IF

	IF (Strncmp(cmd, 'WAGO_DALI_CENTRAL ', 18) = TRUE) THEN
		p1 := GET_PARAM_DINT(cmd, 1);
		p2 := GET_PARAM_DINT(cmd, 2);
		DALIShowShortAdr(xCentr_ON := FALSE, xCentr_OFF := FALSE);
		IF (p2 = 1) THEN
			DALIShowShortAdr(xCentr_ON := TRUE);
		ELSE
			DALIShowShortAdr(xCentr_OFF := TRUE);
		END_IF
	END_IF

	IF (Strncmp(cmd, 'WAGO_DALI_BLINK ', 16) = TRUE) THEN
		p1 := GET_PARAM_DINT(cmd, 1);
		p2 := GET_PARAM_DINT(cmd, 2); (* address *)
		p3 := GET_PARAM_DINT(cmd, 3); (* group? *)
		p4 := GET_PARAM_DINT(cmd, 4); (* blink time *)
		DALIShowShortAdr(xBlink := FALSE);
		DALIShowShortAdr(xBlink := TRUE, bAddress := DINT_TO_BYTE(p2), bBlinkTime := DINT_TO_BYTE(p4), xGroup := DINT_TO_BOOL(p3));
	END_IF

	IF (Strncmp(cmd, 'WAGO_DALI_BLINK_STOP ', 21) = TRUE) THEN
		p1 := GET_PARAM_DINT(cmd, 1);
		DALIShowShortAdr(xBlink_OFF := FALSE);
		DALIShowShortAdr(xBlink_OFF := TRUE);
	END_IF

	IF (Strncmp(cmd, 'WAGO_DALI_SET_DEVICE_CONFIG ', 28) = TRUE) THEN
		p1 := GET_PARAM_DINT(cmd, 1);
		p2 := GET_PARAM_DINT(cmd, 2); (* device address *)
		p3 := GET_PARAM_DINT(cmd, 3); (* fade rate *)
		p4 := GET_PARAM_DINT(cmd, 4); (* fade time *)
		p5 := GET_PARAM_DINT(cmd, 5); (* max level *)
		p6 := GET_PARAM_DINT(cmd, 6); (* min level *)
		p7 := GET_PARAM_DINT(cmd, 7); (* system failure level *)
		p8 := GET_PARAM_DINT(cmd, 8); (* power on level *)
		DALIConfigDevice(xSetConfig := FALSE);
		DALIConfigDevice(xSetConfig := TRUE, bAddress := DINT_TO_BYTE(p2),
					bFade_Rate := DINT_TO_BYTE(p3), bFade_Time := DINT_TO_BYTE(p4),
					bMax_Level := DINT_TO_BYTE(p5), bMin_Level := DINT_TO_BYTE(p6),
					bSystem_Failure_Level := DINT_TO_BYTE(p7), bPower_On_Level := DINT_TO_BYTE(p8));
	END_IF

	IF (Strncmp(cmd, 'WAGO_DALI_ADDRESSING_NEW ', 25) = TRUE) THEN
		p1 := GET_PARAM_DINT(cmd, 1);
		p2 := GET_PARAM_DINT(cmd, 2); (* reset? *)
		DALIConfigShortAddress(xNewAddressing := FALSE);
		DALIConfigShortAddress(xNewAddressing := TRUE, xReset := DINT_TO_BOOL(p2), xSwitchAtAddressing := TRUE);
		DALIConfigShortAddress(xNewAddressing := FALSE); (* double click *)
		DALIConfigShortAddress(xNewAddressing := TRUE, xReset := DINT_TO_BOOL(p2), xSwitchAtAddressing := TRUE);
		replaceAddr := FALSE;
		extendedAddr := FALSE;
		newAddressing := TRUE;
		delAddressing := FALSE;
		resetAddr := DINT_TO_BOOL(p2);
		DaliSendAction := 99; (* addressing in progress *)
	END_IF

	IF (Strncmp(cmd, 'WAGO_DALI_ADDRESSING_ADD ', 25) = TRUE) THEN
		p1 := GET_PARAM_DINT(cmd, 1);
		DALIConfigShortAddress(xExtendedAddressing := FALSE);
		DALIConfigShortAddress(xExtendedAddressing := TRUE, xSwitchAtAddressing := TRUE);
		replaceAddr := FALSE;
		extendedAddr := TRUE;
		newAddressing := FALSE;
		resetAddr := FALSE;
		delAddressing := FALSE;
		DaliSendAction := 99; (* addressing in progress *)
	END_IF

	IF (Strncmp(cmd, 'WAGO_DALI_ADDRESSING_STATUS ', 28) = TRUE) THEN
		p1 := GET_PARAM_DINT(cmd, 1);
		DaliSendAction := 98; (* addressing in progress *)
	END_IF

	IF (Strncmp(cmd, 'WAGO_DALI_ADDRESSING_CHANGE ', 28) = TRUE) THEN
		p1 := GET_PARAM_DINT(cmd, 1);
		p2 := GET_PARAM_DINT(cmd, 2); (* old address *)
		p3 := GET_PARAM_DINT(cmd, 3); (* new address *)
		oldAddr := DINT_TO_BYTE(p2);
		newAddr := DINT_TO_BYTE(p3);
		DALIConfigShortAddress(xReplaceShortAddress := FALSE);
		DALIConfigShortAddress(xReplaceShortAddress := TRUE, bOldShortAddress := oldAddr, bNewShortAddress := newAddr);
		replaceAddr := TRUE;
		extendedAddr := FALSE;
		newAddressing := FALSE;
		resetAddr := FALSE;
		delAddressing := FALSE;
		DaliSendAction := 99; (* addressing in progress *)
	END_IF

	IF (Strncmp(cmd, 'WAGO_DALI_ADDRESSING_DEL ', 25) = TRUE) THEN
		p1 := GET_PARAM_DINT(cmd, 1);
		p2 := GET_PARAM_DINT(cmd, 2); (* address to delete *)
		delAddr := DINT_TO_BYTE(p2);
		DALIConfigShortAddress(xDeleteShortAddress := FALSE);
		DALIConfigShortAddress(xDeleteShortAddress := TRUE, bDeleteShortAddress := delAddr);
		replaceAddr := TRUE;
		extendedAddr := FALSE;
		newAddressing := FALSE;
		resetAddr := FALSE;
		delAddressing := TRUE;
		DaliSendAction := 99; (* addressing in progress *)
	END_IF

END_IF

CASE DaliSendAction OF
(*
1: (* WAGO_DALI_GET_ADDR *)
	IF (DALIShowShortAdr.xReady = TRUE) THEN
		cmd := 'WAGO_DALI_GET_ADDR ';
		cmd := CONCAT(cmd, WORD_TO_STRB(DALIShowShortAdr.wShortAddress_16_1));
		cmd := CONCAT(cmd, WORD_TO_STRB(DALIShowShortAdr.wShortAddress_32_17));
		cmd := CONCAT(cmd, WORD_TO_STRB(DALIShowShortAdr.wShortAddress_48_33));
		cmd := CONCAT(cmd, WORD_TO_STRB(DALIShowShortAdr.wShortAddress_64_49));
		start_send := TRUE;
		DaliSendAction := 0;
	ELSE
		DALIShowShortAdr(xQuery := TRUE);
	END_IF
*)
1: (* WAGO_DALI_GET_ADDR *)
	IF (dali_master = FALSE) THEN
		addr_1_16 := SHL(DaliMasterAdv.bByte_3, 8) + DaliMasterAdv.bByte_1;
		addr_17_32 := SHL(DaliMasterAdv.bByte_5, 8) + DaliMasterAdv.bByte_4;
		dali_master := TRUE;
		DALIMasterAdv(xStartDaliMaster := dali_master, iCommand := 507);
		DaliSendAction := 111;
	ELSE
		DaliMasterAdv(xStartDaliMaster := dali_master);
	END_IF
111: (* WAGO_DALI_GET_ADDR bis *)
	IF (dali_master = FALSE) THEN
		cmd := 'WAGO_DALI_GET_ADDR ';
		cmd := CONCAT(cmd, WORD_TO_STRB(addr_1_16));
		cmd := CONCAT(cmd, WORD_TO_STRB(addr_17_32));
		cmd := CONCAT(cmd, WORD_TO_STRB( SHL(DaliMasterAdv.bByte_3, 8) + DaliMasterAdv.bByte_1 ));
		cmd := CONCAT(cmd, WORD_TO_STRB( SHL(DaliMasterAdv.bByte_5, 8) + DaliMasterAdv.bByte_4 ));
		start_send := TRUE;
		DaliSendAction := 0;
	ELSE
		DaliMasterAdv(xStartDaliMaster := dali_master);
	END_IF
2: (* WAGO_DALI_GET_DEVICE_INFO *)
	IF (DALIConfigDevice.xReady = TRUE) THEN
		cmd := 'WAGO_DALI_GET_DEVICE_INFO ';
		cmd := CONCAT(cmd, WORD_TO_STRING(DALIConfigDevice.bFadeRate));
		cmd := CONCAT(cmd, ' ');
		cmd := CONCAT(cmd, WORD_TO_STRING(DALIConfigDevice.bFadeTime));
		cmd := CONCAT(cmd, ' ');
		cmd := CONCAT(cmd, WORD_TO_STRING(DALIConfigDevice.bMaxLevel));
		cmd := CONCAT(cmd, ' ');
		cmd := CONCAT(cmd, WORD_TO_STRING(DALIConfigDevice.bMinLevel));
		cmd := CONCAT(cmd, ' ');
		cmd := CONCAT(cmd, WORD_TO_STRING(DALIConfigDevice.bSystemFailureLevel));
		cmd := CONCAT(cmd, ' ');
		cmd := CONCAT(cmd, WORD_TO_STRING(DALIConfigDevice.bPowerOnLevel));
		start_send := TRUE;
		DaliSendAction := 0;
	ELSE
		DALIConfigDevice(xQuery := TRUE);
	END_IF
3: (* WAGO_DALI_GET_DEVICE_GROUP *)
	IF (dali_master = FALSE) THEN
		groups_cmd_1_8 := DaliMaster.bQueryValue;
		dali_master := TRUE;
		DALIMaster(xStartDaliMaster := dali_master, iCommand := 193, bAddress := group_address);
		DaliSendAction := 4;
	ELSE
		DaliMaster(xStartDaliMaster := dali_master);
	END_IF
4: (* WAGO_DALI_GET_DEVICE_GROUP bis *)
	IF (dali_master = FALSE) THEN
		cmd := 'WAGO_DALI_GET_DEVICE_GROUP ';
		cmd := CONCAT(cmd, BYTE_TO_STRING(group_address));
		cmd := CONCAT(cmd, ' ');
		cmd := CONCAT(cmd, WORD_TO_STRB( SHL(DaliMaster.bQueryValue, 8) + groups_cmd_1_8 ));
		start_send := TRUE;
		DaliSendAction := 0;
	ELSE
		DaliMaster(xStartDaliMaster := dali_master);
	END_IF
5: (* WAGO_DALI_DEVICE_ADD_GROUP *)
	IF (dali_master = FALSE) THEN
		cmd := 'WAGO_DALI_DEVICE_ADD_GROUP 1';
		start_send := TRUE;
		DaliSendAction := 0;
	ELSE
		DALIMasterAdv(xStartDaliMaster := dali_master);
	END_IF
6: (* WAGO_DALI_DEVICE_DEL_GROUP *)
	IF (dali_master = FALSE) THEN
		cmd := 'WAGO_DALI_DEVICE_DEL_GROUP 1';
		start_send := TRUE;
		DaliSendAction := 0;
	ELSE
		DALIMasterAdv(xStartDaliMaster := dali_master);
	END_IF
98: (* WAGO_DALI_ADDRESSING_STATUS *)
	IF (DALIConfigShortAddress.xReady = TRUE) THEN
		cmd := 'WAGO_DALI_ADDRESSING_STATUS 1';
		start_send := TRUE;
		DaliSendAction := 0;
	ELSE
		cmd := 'WAGO_DALI_ADDRESSING_STATUS 0';
		start_send := TRUE;
		DaliSendAction := 99;
		DALIConfigShortAddress(xNewAddressing := newAddressing, xExtendedAddressing := extendedAddr,
							   xReset := resetAddr, xSwitchAtAddressing := TRUE,
							   xReplaceShortAddress := replaceAddr, bOldShortAddress := oldAddr, bNewShortAddress := newAddr,
							   xDeleteShortAddress := delAddressing, bDeleteShortAddress := delAddr);
	END_IF
99: (* Addressing in progress *)
		DALIConfigShortAddress(xNewAddressing := newAddressing, xExtendedAddressing := extendedAddr,
							   xReset := resetAddr, xSwitchAtAddressing := TRUE,
							   xReplaceShortAddress := replaceAddr, bOldShortAddress := oldAddr, bNewShortAddress := newAddr,
							   xDeleteShortAddress := delAddressing, bDeleteShortAddress := delAddr);
END_CASE

IF (DaliSend = TRUE) THEN
	IF (dmx_read_addr > 0) THEN

		cmd := 'WAGO_DALI_GET ';
		IF (abDMX_Values[dmx_read_addr] < 1) THEN
			cmd := CONCAT(cmd, '0 ');
		ELSE
			cmd := CONCAT(cmd, '1 ');
		END_IF
		cmd := CONCAT(cmd, ITOA(BYTE_TO_INT(abDMX_Values[dmx_read_addr] * 100 / 255)));
		start_send := TRUE;
		DaliSend := FALSE;
	ELSE
		IF Config.CONFIG_DALI = TRUE THEN
			IF (DALIDimmValue.xReady = TRUE) THEN
				cmd := 'WAGO_DALI_GET ';
				cmd := CONCAT(cmd, ITOA(BOOL_TO_INT(DALIDimmValue.xStatus)));
				cmd := CONCAT(cmd, ' ');
				cmd := CONCAT(cmd, ITOA(BYTE_TO_INT(DALIDimmValue.bDimmValue)));
				start_send := TRUE;
				DaliSend := FALSE;
			ELSE
				DALIDimmValue(xEnable := TRUE, bShortAddress := DINT_TO_BYTE(p2), tCycleTime := t#1s);
			END_IF
		ELSE
			cmd := 'WAGO_DALI_GET ';
			IF dali_group = TRUE THEN
				IF DaliSendValueGrp647[daliShortAddr].rActualLevel = 0 THEN
					cmd := CONCAT(cmd, '0');
				ELSE
					cmd := CONCAT(cmd, '1');
				END_IF
				cmd := CONCAT(cmd, ' ');
				cmd := CONCAT(cmd, ITOA(REAL_TO_INT(DaliSendValueGrp647[daliShortAddr].rActualLevel)));
			ELSE
				IF DaliSendValue647[daliShortAddr].rActualLevel = 0 THEN
					cmd := CONCAT(cmd, '0');
				ELSE
					cmd := CONCAT(cmd, '1');
				END_IF
				cmd := CONCAT(cmd, ' ');
				cmd := CONCAT(cmd, ITOA(REAL_TO_INT(DaliSendValue647[daliShortAddr].rActualLevel)));
			END_IF
			cmd := CONCAT(cmd, ' ');
			cmd := CONCAT(cmd, ITOA(BYTE_TO_INT(DALIDimmValue.bDimmValue)));
			start_send := TRUE;
			DaliSend := FALSE;
		END_IF
	END_IF
END_IF

IF (HEARTBEAT_TIMER.Q = TRUE) THEN
	(* We lost the connection with the server *)
	(* The wago is now in standalone mode *)
	HEARTBEAT := FALSE;

	LedMode := 1;
ELSE
	HEARTBEAT := TRUE;
END_IF
END_PROGRAM

(* POU EthernetServer_FB, ST *)
FUNCTION_BLOCK EthernetServer_FB
(************************************************************)
(* ETHERNET_SERVER		                          		    *)
(* Ver. 1.0   	                                         	*)
(* Date:  10.02.2003					         	 		*)
(* Author:  Volker Begemann                            		*)
(************************************************************)
VAR_INPUT
	xOPEN_SERVER		:	BOOL;				(* Set TRUE to enable function block			*)
	wPORT					:	WORD;				(* Port number											*)
	xTCP_PROTOCOL		:	BOOL;				(* TRUE => TCP; FALSE => UDP						*)
	tTIMEOUT				:	TIME:=t#20s;	(* Watchdog timeout value (seconds)				*)
	iBYTES_TO_SEND		:	INT;				(* Number of bytes to transmit					*)
	ptSEND_BUFFER		:	POINTER TO ARRAY[1..1500] OF BYTE;		(* Transmit Buffer	*)
END_VAR
VAR_IN_OUT
	xSTART_SEND:		BOOL;						(* Set TRUE to initiate data transmittal, will be	*)
														(* reset FALSE when transmittal is completed 		*)
(* 	utRECEIVE_BUFFER:	typEthernetBuffer;	(* Receive Buffer *) *)
	ptRECV_BUFFER		:	POINTER TO ARRAY[1..1500] OF BYTE;		(* Receive Buffer	*)
END_VAR
VAR_OUTPUT
	utERROR					:	ETH_ERROR;	(* See ETH_ERROR datatype in ETHERNET.LIB	*)
													(* for error codes and definitions			*)
	xSERVER_OPEN:			BOOL;				(* TRUE if socket connection made			*)
	wSOCKET:					WORD;				(* Socket connection number					*)
	bDataReceived: 		BOOL := FALSE;
	iBYTES_RECEIVED: INT; (* Number of bytes received *)
END_VAR
VAR
	i: INT;
	CloseState:			INT;
	EthernetOpen:		ETHERNET_SERVER_OPEN;
	EthernetClose:		ETHERNET_SERVER_CLOSE;
	EthernetWrite:		ETHERNET_WRITE;
	EthernetRead:		ETHERNET_READ;
	GetConfig:			ETHERNET_GET_NETWORK_CONFIG;
	EthernetBuffer:	ARRAY[1..1500] OF BYTE;
	Status:				WORD:=0;
	client_SRC_PORT:	WORD;
	watchdog_timer1:	TON;
	client_SRC_IP:		DWORD;
END_VAR
IF xOPEN_SERVER THEN
	watchdog_timer1(IN:=TRUE , PT:=tTIMEOUT );

	IF watchdog_timer1.q THEN
		watchdog_timer1(IN:=FALSE , PT:=tTIMEOUT );
		EthernetClose(EN:= 1, SOCKET:= EthernetOpen.SOCKET);
		EthernetClose(EN:= 0, SOCKET:= 0);
		Status := 0; (* Try to open the server *)
	END_IF

	CASE Status OF
		0:
			GetConfig(EN:=FALSE );
			GetConfig(EN:=TRUE );
			utERROR		:=	0;
			wSocket		:=	0;
			CloseState	:=	0;
			status		:=	1;
		1:
			GetConfig(EN:=TRUE );
			IF GetConfig.ENO THEN
				IF GetConfig.IP_ADR<>0 THEN
					status:=4;
					EthernetOpen (EN:=0);
					EthernetRead(EN:= 0, SOCKET:=0 ,  DATA:=EthernetBuffer );
					EthernetClose(EN:= 0);
				ELSE
					status:=0;
				END_IF
			END_IF
		4: 	(* try to open a socket*)
			IF xTCP_PROTOCOL THEN
				EthernetOpen(EN:=1 , TYP:=SOCK_STREAM, PROTO := IPPROTO_TCP, PORT := wPort);
			ELSE
				EthernetOpen(EN:=1 , TYP:=SOCK_DGRAM, PROTO := IPPROTO_UDP, PORT := wPort);
			END_IF
			IF ((EthernetOpen.ERROR = 0) AND (EthernetOpen.ENO = 1)) THEN
				Status  := 10; (* socket created, wait for data to process *)
				EthernetOpen (EN:=0);
				xServer_open:=TRUE;
				wSocket:=EthernetOpen.socket;
			ELSE
				Status := 0; 	(* socket not available, try it again *)
				EthernetOpen (EN:=0);
				xServer_open:=FALSE;
				wSocket:=0;
			END_IF;

		10: 	(* Wait for data to process *)
			(* Monitor ethernet port for new data *)
			bDataReceived	:= FALSE;
	 		EthernetRead(	EN:= 1, SOCKET:=EthernetOpen.SOCKET, DATA:=EthernetBuffer);
			EthernetRead(	EN:= 0, SOCKET:=0, DATA:=EthernetBuffer);

			IF(EthernetRead.ERROR<>0) THEN  			(* Error reading the socket, close it *)
				Status	:=	40;
			ELSIF (EthernetRead.LEN_OUT <>0) THEN  (* Process the data received via the ethernet port *)
				client_SRC_IP		:=	EthernetRead.SRC_IP;
				client_SRC_PORT	:=	EthernetRead.SRC_PORT;
				ptRECV_BUFFER^		:= EthernetBuffer;
				bDataReceived		:= TRUE;
				iBYTES_RECEIVED		:= EthernetRead.LEN_OUT;
				watchdog_timer1(IN:=FALSE, PT:=tTIMEOUT );
			ELSIF (iBytes_TO_SEND > 0 AND xSTART_SEND) THEN  (* Process the data received *)
				EthernetWrite(EN:= 0, DATA:=EthernetBuffer);
				status	:=	30;
			END_IF

		30: 	(* Process the data to send *)
			EthernetBuffer :=ptSEND_BUFFER^;
			(* Send data in transmit buffer out ethernet port *)
			IF xTCP_PROTOCOL THEN
					EthernetWrite(	EN:= 1,
								SOCKET:= EthernetOpen.SOCKET,
								LEN_IN:=iBYTES_TO_SEND,
								DATA:=EthernetBuffer );
			ELSE
				IF client_SRC_IP>0 AND client_SRC_PORT>0 THEN
					EthernetWrite(EN:=1, SOCKET:=EthernetOpen.SOCKET , LEN_IN:=iBYTES_TO_SENd , DST_IP:=client_SRC_IP,DST_PORT:=client_SRC_PORT,DATA:=EthernetBuffer );
				ELSE
					status:=10;
				END_IF
			END_IF

			IF EthernetWrite.eno THEN
				IF(EthernetWrite.ERROR <>0) THEN
					Status:=40;(* Error writing to the socket, close it *)
				ELSE
					Status:=10; (* Comms complete, read more data *)
				END_IF;
				xStart_send:=FALSE;
			END_IF
		40:	(* Close the server *)
			EthernetClose(EN:= 1, SOCKET:= EthernetOpen.SOCKET);
			IF EthernetClose.eno THEN
				EthernetClose(EN:= 0);
				xOPEN_SERVER:=FALSE;
				utERROR:=0;
				wSocket:=0;
				Status := 0; (* Try to open the server again *)
			END_IF

	END_CASE;
ELSE
	CASE CloseState OF
	0:
		EthernetClose(EN:= 0);
		EthernetClose(EN:= 1, SOCKET:= EthernetOpen.SOCKET);
		CloseState:=1;
	1:
		EthernetClose(EN:= 1, SOCKET:= EthernetOpen.SOCKET);
		IF EthernetClose.eno THEN
			EthernetClose(EN:= 0);
			CloseState:=2;
		END_IF
	2:
		xOPEN_SERVER:=FALSE;
		utERROR:=0;
		wSocket:=0;
	END_CASE
END_IF
END_FUNCTION_BLOCK

(* POU Strncmp, ST *)
FUNCTION Strncmp : BOOL
VAR_INPUT
	str1: STRING;
	str2: STRING;
	n: BYTE;
END_VAR
VAR
	tmp1: POINTER TO ARRAY[0..255] OF BYTE;
	tmp2: POINTER TO ARRAY[0..255] OF BYTE;
	i: BYTE;
END_VAR
tmp1 := ADR(str1);
tmp2 := ADR(str2);

Strncmp := TRUE;

FOR i := 0 TO n - 1 DO
	IF (tmp1^[i] <> tmp2^[i]) THEN
		Strncmp := FALSE;
		i := n;
	END_IF
END_FOR
END_FUNCTION

(* POU GET_PARAM_DINT, ST *)
FUNCTION GET_PARAM_DINT : DINT
VAR_INPUT
	str: STRING;
	pos: BYTE;
END_VAR
VAR
	i: BYTE;
	j: BYTE;
	mult : DWORD;
	dec : DWORD;
	p: INT;
	tmp: POINTER TO ARRAY[0..255] OF BYTE;
	val: DINT;
	neg: BOOL := FALSE;
	found: INT;
END_VAR
(* cut before the value we want *)
FOR i := 1 TO pos DO
	found := FIND(str, ' ');
	IF found = 0 THEN
		GET_PARAM_DINT := 0;
		RETURN;
	END_IF
	str := DELETE(str, found, 1);
END_FOR

(* cut after the value we want *)
p := FIND(str, ' ');
IF (p > 0) THEN
	str := LEFT(str, p - 1);
END_IF

(* Convert the value *)
tmp := ADR(str);

IF (Strncmp(str, '-', 1) = TRUE) THEN
	neg := TRUE;
	str := DELETE(str, 1, 1);
END_IF

val := 0;
FOR i := 0 TO INT_TO_BYTE(LEN(str) - 1) DO
	dec := 1;
	FOR j := 2 TO INT_TO_BYTE(LEN(str) - i) DO
		dec := dec * 10;
	END_FOR

	mult := tmp^[i] - 16#30;
	mult := mult * dec;
	val := val + mult;

END_FOR

IF (neg = TRUE) THEN
	GET_PARAM_DINT := 0 - val;
ELSE
	GET_PARAM_DINT := val;
END_IF
END_FUNCTION

(* POU VOLET, ST *)
FUNCTION_BLOCK VOLET
VAR
	sens: BOOL;
	imp: TP;
	mode: VOLET_MODE;
END_VAR
VAR_INPUT
	IN: BOOL;
	IMPULSE: BOOL;
END_VAR
VAR_OUTPUT
	MONTE: BOOL;
	DESCENTE:BOOL;
END_VAR
(* Volet *)

IF IMPULSE = FALSE THEN
	(* Normal mode *)
	IF (MONTE = TRUE OR DESCENTE = TRUE) THEN
		MONTE := FALSE;
		DESCENTE := FALSE;
	ELSE

		IF IN = TRUE THEN
			IF sens = TRUE THEN
				sens := FALSE;
			ELSE
				sens := TRUE;
			END_IF;

			IF sens = TRUE THEN
				(*monte*)
				DESCENTE := FALSE;
				MONTE := TRUE;
			ELSE
				MONTE := FALSE;
				DESCENTE := TRUE;
			END_IF;
		END_IF

	END_IF
ELSE
	(* impulse mode *)
	imp(IN := FALSE, PT:= impulse_time);

	IF mode = IMP_STOP THEN
		MONTE := imp.Q;
		DESCENTE := imp.Q;
		IF imp.Q = FALSE THEN
			mode := VOLET_STOP;
		END_IF;
	END_IF;
	IF mode = IMP_UP THEN
		MONTE := imp.Q;
		DESCENTE := FALSE;
		IF imp.Q = FALSE THEN
			mode := VOLET_UP;
		END_IF;
	END_IF;
	IF mode = IMP_DOWN THEN
		MONTE := FALSE;
		DESCENTE := imp.Q;
		IF imp.Q = FALSE THEN
			mode := VOLET_DOWN;
		END_IF;
	END_IF;

	IF mode = VOLET_UP OR mode = VOLET_DOWN THEN
		IF IN = TRUE THEN
			imp(IN := TRUE, PT:= impulse_time);
			mode := IMP_STOP;
		END_IF;
	ELSE
		IF IN = TRUE THEN
			IF sens = TRUE THEN
				sens := FALSE;
			ELSE
				sens := TRUE;
			END_IF;

			IF sens = TRUE THEN
				imp(IN := TRUE, PT:= impulse_time);
				mode := IMP_UP;
			ELSE
				imp(IN := TRUE, PT:= impulse_time);
				mode := IMP_DOWN;
			END_IF;
		END_IF;
	END_IF;
END_IF;
END_FUNCTION_BLOCK

(* POU ITOA, ST *)
FUNCTION ITOA : STRING
VAR_INPUT
	VAL: INT;
END_VAR
VAR
	tmp: INT;
	conv: INT;
END_VAR
(* Convert a byte to string *)

IF (VAL < 0) THEN
	tmp := -VAL;
ELSE
	tmp := VAL;
END_IF

IF (tmp = 0) THEN
	ITOA := ASCIIBYTE_TO_STRING(0 + 16#30);
END_IF

WHILE (tmp > 0) DO
	conv := tmp MOD 10;
	tmp := tmp / 10;
	ITOA := INSERT(ITOA, ASCIIBYTE_TO_STRING(INT_TO_BYTE(conv) + 16#30), 0);
END_WHILE

IF (VAL < 0) THEN
	ITOA := INSERT(ITOA, '-', 0);
END_IF
END_FUNCTION

(* POU DMX, FBD *)
PROGRAM DMX
VAR
	DMX_Master				: FbDMX_StageProfi;
		Enable				: BOOL := TRUE ;
		PortNumber			: WORD := 10001;
		FirstChannel		: WORD := 1;
		NumberOfChannels	: BYTE := 255;
		Ready				: BOOL;
		Connect				: BOOL;
		ErrorCode			: DINT;
		ErrorWatchdog		: BOOL;
END_VAR
VAR_INPUT RETAIN
		IPaddress			: STRING(16) := '192.168.1.120';
END_VAR
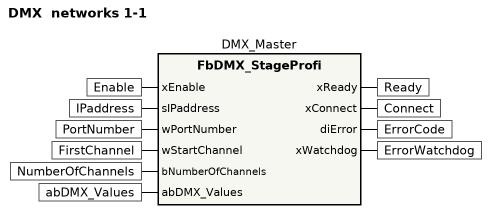
_FBD_ (* Function Block Diagram *)
NETWORK 1
	DMX_Master:FbDMX_StageProfi(xEnable: Enable, sIPaddress: IPaddress, wPortNumber: PortNumber, wStartChannel: FirstChannel, bNumberOfChannels: NumberOfChannels, abDMX_Values: abDMX_Values, xConnect => Connect, diError => ErrorCode, xWatchdog => ErrorWatchdog) => Ready
_END_FBD_
(* the same logic as Structured Text *)
(* Network 1 *)
DMX_Master(xEnable := Enable, sIPaddress := IPaddress, wPortNumber := PortNumber, wStartChannel := FirstChannel, bNumberOfChannels := NumberOfChannels, abDMX_Values := abDMX_Values);
Connect := DMX_Master.xConnect;
ErrorCode := DMX_Master.diError;
ErrorWatchdog := DMX_Master.xWatchdog;
Ready := DMX_Master.xReady;
END_PROGRAM

(* POU SetOutput, ST *)
FUNCTION SetOutput : BOOL
VAR_INPUT
	bit_offset: UINT;
	val: BOOL;
END_VAR
VAR
END_VAR
(* Set the bit in OutArrState Array *)

IF (val = TRUE) THEN
	OutArrState[bit_offset / 8] := OutArrState[bit_offset / 8] OR SHL(BYTE#01, bit_offset MOD 8);
ELSE
	OutArrState[bit_offset / 8] := OutArrState[bit_offset / 8] AND NOT SHL(BYTE#01, bit_offset MOD 8);
END_IF

SetOutput := TRUE;
END_FUNCTION

(* POU WORD_TO_STRB, ST *)
FUNCTION WORD_TO_STRB : STRING(16)
VAR_INPUT
	IN : WORD;
END_VAR
VAR
	pt : POINTER TO BYTE;
	i: INT;
END_VAR
pt := ADR(WORD_TO_STRB);

FOR i := 1 TO 16 DO
	pt^:= BOOL_TO_BYTE(in.0) + 48;
	in := SHR(in,1);
	pt := pt + 1;
END_FOR;

pt^ := 0;
END_FUNCTION

(* POU ManageOutput, ST *)
PROGRAM ManageOutput
VAR
	cpt: INT;
	tmp: INT;
	_light: LIGHT;
	in: BOOL;
END_VAR
(* Set all outputs when in standalone mode *)

(* Get the address of the first digital output *)
FOR cpt := 0 TO 512 DO

	CASE output_type[cpt] OF
	NONE: (* Do nothing *);
	TELERUPTEUR:
		tmp := cpt;
		IF (output_addr[cpt].SameAs >= 0) THEN
			tmp := output_addr[cpt].SameAs;
		END_IF
		IF (event[cpt].ON = TRUE) THEN
			_light(IN := FALSE, STATE := BYTE_TO_BOOL(SHR(lights[tmp / 8], tmp MOD 8) AND 16#01));
			_light(IN := TRUE, STATE := BYTE_TO_BOOL(SHR(lights[tmp / 8], tmp MOD 8) AND 16#01));
			SetOutput(output_addr[tmp].ADDR1 + start_addr_out, _light.OUT);

			(* set old state *)
			IF (_light.OUT = TRUE) THEN
				lights[tmp / 8] := lights[tmp / 8] OR SHL(BYTE#1, tmp MOD 8);
			ELSE
				lights[tmp / 8] := lights[tmp / 8] AND NOT SHL(BYTE#1, tmp MOD 8);
			END_IF
		END_IF
	DIRECT:
		tmp := cpt;
		IF (output_addr[cpt].SameAs >= 0) THEN
			tmp := output_addr[cpt].SameAs;
		END_IF
		in := GetInput(cpt + start_addr_in);
		SetOutput(output_addr[tmp].ADDR1 + start_addr_out, in);
	VOLET:
		tmp := cpt;
		IF (output_addr[cpt].SameAs >= 0) THEN
			tmp := output_addr[cpt].SameAs;
		END_IF
		IF (event[cpt].ON = TRUE) THEN
			volets[tmp](IN := TRUE, IMPULSE := FALSE);
			SetOutput(output_addr[tmp].ADDR1 + start_addr_out, volets[tmp].MONTE);
			SetOutput(output_addr[tmp].ADDR2 + start_addr_out, volets[tmp].DESCENTE);
		END_IF
	VOLET_IMPULSE:
		tmp := cpt;
		IF (output_addr[cpt].SameAs >= 0) THEN
			tmp := output_addr[cpt].SameAs;
		END_IF
		IF (event[cpt].ON = TRUE) THEN
			volets[tmp](IN := TRUE, IMPULSE := TRUE);
		ELSE
			volets[tmp](IN := FALSE, IMPULSE := TRUE);
		END_IF
		SetOutput(output_addr[tmp].ADDR1 + start_addr_out, volets[tmp].MONTE);
		SetOutput(output_addr[tmp].ADDR2 + start_addr_out, volets[tmp].DESCENTE);
	TELERUPTEUR_DALI:
		tmp := cpt;
		IF (output_addr[cpt].SameAs >= 0) THEN
			tmp := output_addr[cpt].SameAs;
		END_IF
		IF (event[cpt].ON = TRUE) THEN
			_light(IN := FALSE, STATE := BYTE_TO_BOOL(SHR(lights[tmp / 8], tmp MOD 8) AND 16#01));
			_light(IN := TRUE, STATE := BYTE_TO_BOOL(SHR(lights[tmp / 8], tmp MOD 8) AND 16#01));

			IF (output_addr[tmp].ADDR2 > 99) THEN
				IF (_light.OUT = TRUE) THEN
					abDMX_Values[WORD_TO_BYTE(output_addr[tmp].ADDR2 - 100)] := 255;
				ELSE
					abDMX_Values[WORD_TO_BYTE(output_addr[tmp].ADDR2 - 100)] := 0;
				END_IF
			ELSE
				Dali_switch(bAddress := WORD_TO_BYTE(output_addr[tmp].ADDR2), xGroup := FALSE, xButton := FALSE);
				IF (_light.OUT = TRUE) THEN
					Dali_switch(bAddress := WORD_TO_BYTE(output_addr[tmp].ADDR2), xGroup := FALSE, bDimmLevel := 100,
						bFadeTime := 1, xButton := TRUE);
				ELSE
					Dali_switch(bAddress := WORD_TO_BYTE(output_addr[tmp].ADDR2), xGroup := FALSE, bDimmLevel := 0,
						bFadeTime := 1, xButton := TRUE);
				END_IF
			END_IF

			(* set old state *)
			IF (_light.OUT = TRUE) THEN
				lights[tmp / 8] := lights[tmp / 8] OR SHL(BYTE#1, tmp MOD 8);
			ELSE
				lights[tmp / 8] := lights[tmp / 8] AND NOT SHL(BYTE#1, tmp MOD 8);
			END_IF
		END_IF
	TELERUPTEUR_DALI_GROUP:
		tmp := cpt;
		IF (output_addr[cpt].SameAs >= 0) THEN
			tmp := output_addr[cpt].SameAs;
		END_IF
		IF (event[cpt].ON = TRUE) THEN
			_light(IN := FALSE, STATE := BYTE_TO_BOOL(SHR(lights[tmp / 8], tmp MOD 8) AND 16#01));
			_light(IN := TRUE, STATE := BYTE_TO_BOOL(SHR(lights[tmp / 8], tmp MOD 8) AND 16#01));
			Dali_switch(bAddress := output_addr[tmp].ADDR2, xGroup := TRUE, xButton := FALSE);
			IF (_light.OUT = TRUE) THEN
				Dali_switch(bAddress := output_addr[tmp].ADDR2, xGroup := TRUE, bDimmLevel := 100,
					bFadeTime := 1, xButton := TRUE);
			ELSE
				Dali_switch(bAddress := output_addr[tmp].ADDR2, xGroup := TRUE, bDimmLevel := 0,
					bFadeTime := 1, xButton := TRUE);
			END_IF

			(* set old state *)
			IF (_light.OUT = TRUE) THEN
				lights[tmp / 8] := lights[tmp / 8] OR SHL(BYTE#1, tmp MOD 8);
			ELSE
				lights[tmp / 8] := lights[tmp / 8] AND NOT SHL(BYTE#1, tmp MOD 8);
			END_IF
		END_IF
	END_CASE
END_FOR
END_PROGRAM

(* POU LIGHT, ST *)
FUNCTION_BLOCK LIGHT
VAR
	TRIG: R_TRIG;
	light: BOOL;
END_VAR
VAR_INPUT
	IN: BOOL;
	STATE: BOOL;
END_VAR
VAR_OUTPUT
	OUT: BOOL;
END_VAR
(* telerupteur *)

TRIG(CLK := IN);
light := TRIG.Q;

OUT := STATE;

IF light = TRUE THEN
	IF OUT = TRUE THEN
		OUT := FALSE;
	ELSE
		OUT := TRUE;
	END_IF;
END_IF;
END_FUNCTION_BLOCK

(* POU DALI/DaliPrg647, ST *)
PROGRAM DaliPrg647
VAR
	i: INT;
	iDali: INT;
	daliFeedback: BYTE;

	init_dali: BOOL := FALSE;
	startCsvRead: BOOL := TRUE;

	(* DALI 753-647 *)
	DALIMaster647: FbMaster753_647;

	DALI647_InReal AT %IB0: ARRAY[0..23] OF BYTE;
	DALI647_OutReal AT %QB0: ARRAY[0..23] OF BYTE;

END_VAR
(*
	This needs to run on every cycle to update DALI status.
	It is needed by the 647 module FB API which is not working as the
	old 641 API. It should stay in the main cycle loop.
*)

(* read the CSV file listing all DALI sensors type and address available on the bus *)
DaliReadCsvFile(xStart := startCsvRead, daliSensors := daliSensors);

(* the master DALI FB *)
DALIMaster647(
	abIn_753_647 := DALI647_InReal,
	bModule_753_647 := 1,
	abOut_753_647 => DALI647_OutReal,
	bFeedback => daliFeedback
);

(* This is for DALI config program *)
PrgDALIConfig;
(*PrgDALIConfigSensorType1;
PrgDALIConfigSensorType2;*)

(* After first cycle, init dali is done *)
IF (init_dali = FALSE) THEN
	init_dali := TRUE;
END_IF

(* instanciate all DALI sensors based on what is declared in the CSV file *)
FOR i := 1 TO MaxDaliSensors DO
	iDali := i - 1;

	(* handle all dali sensors *)
	IF daliSensors[i].SensorType = MultiSensorType1 THEN
		DaliSensorT1[i](
			typMultiSensorType1 := FuTypMultiSensorType1(
				bAddressPresence := daliSensors[i].AddrPresence - 1,
				bAddressLightLevel := daliSensors[i].AddrLightLevel - 1,
				bModule_753_647 := 1
			),
			tOffDelay := daliSensors[i].offDelay
		);
		DaliSensorsInputs[iDali * 12] := DaliSensorT1[i].xPresence;
		netDaliLevels[daliSensors[i].AddrLightLevel - 1] := REAL_TO_WORD(DaliSensorT1[i].rLightLevel);
		DaliSendSensor(i := iDali * 12);
	ELSIF daliSensors[i].SensorType = PushbuttonSensorType1 THEN
		DaliButtonT1[i](
			typPushButtonSensorType1 := FuTypPushButtonSensorType1(
				bAddressButton1 := daliSensors[i].AddrButton1 - 1,
				bAddressButton2 := daliSensors[i].AddrButton2 - 1,
				bAddressButton3 := daliSensors[i].AddrButton3 - 1,
				bAddressButton4 := daliSensors[i].AddrButton4 - 1,
				bModule_753_647 := 1
			),
		);
		DaliSensorsInputs[iDali* 12] := DaliButtonT1[i].xButton1;
		DaliSensorsInputs[iDali * 12 + 1] := DaliButtonT1[i].xButton2;
		DaliSensorsInputs[iDali * 12 + 2] := DaliButtonT1[i].xButton3;
		DaliSensorsInputs[iDali * 12 + 3] := DaliButtonT1[i].xButton4;
		DaliSendSensor(i := iDali * 12);
		DaliSendSensor(i := iDali * 12 + 1);
		DaliSendSensor(i := iDali * 12 + 2);
		DaliSendSensor(i := iDali * 12 + 3);
	ELSIF daliSensors[i].SensorType = MultiSensorType2 THEN
		DaliSensorT2[i](
			typMultiSensorType2 := FuTypMultiSensorType2(
				bAddressPresence := daliSensors[i].AddrPresence - 1,
				bAddressLightLevel := daliSensors[i].AddrLightLevel - 1,
				bAddressRemoteControl := daliSensors[i].AddrRemote - 1,
				bModule_753_647 := 1
			),
			tOffDelay := daliSensors[i].offDelay
		);
		DaliSensorsInputs[iDali * 12] := DaliSensorT2[i].xPresence;
		DaliSensorsInputs[iDali * 12 + 1] := DaliSensorT2[i].xButton1;
		DaliSensorsInputs[iDali * 12 + 2] := DaliSensorT2[i].xButton2;
		DaliSensorsInputs[iDali * 12 + 3] := DaliSensorT2[i].xButton3;
		DaliSensorsInputs[iDali * 12 + 4] := DaliSensorT2[i].xButton4;
		DaliSensorsInputs[iDali * 12 + 5] := DaliSensorT2[i].xButton5;
		DaliSensorsInputs[iDali * 12 + 6] := DaliSensorT2[i].xButton6;
		DaliSensorsInputs[iDali * 12 + 7] := DaliSensorT2[i].xButton7;
		DaliSensorsInputs[iDali * 12 + 8] := DaliSensorT2[i].xButton8;
		DaliSensorsInputs[iDali * 12 + 9] := DaliSensorT2[i].xButton9;
		DaliSensorsInputs[iDali * 12 + 10] := DaliSensorT2[i].xButton10;
		DaliSensorsInputs[iDali * 12 + 11] := DaliSensorT2[i].xButton11;
		netDaliLevels[daliSensors[i].AddrLightLevel - 1] := REAL_TO_WORD(DaliSensorT2[i].rLightLevel);
		DaliSendSensor(i := iDali * 12);
		DaliSendSensor(i := iDali * 12 + 1);
		DaliSendSensor(i := iDali * 12 + 2);
		DaliSendSensor(i := iDali * 12 + 3);
		DaliSendSensor(i := iDali * 12 + 4);
		DaliSendSensor(i := iDali * 12 + 5);
		DaliSendSensor(i := iDali * 12 + 6);
		DaliSendSensor(i := iDali * 12 + 7);
		DaliSendSensor(i := iDali * 12 + 8);
		DaliSendSensor(i := iDali * 12 + 9);
		DaliSendSensor(i := iDali * 12 + 10);
		DaliSendSensor(i := iDali * 12 + 11);
	ELSIF daliSensors[i].SensorType = PushbuttonSensorType2 THEN
		DaliButtonT2[i](
			typPushButtonSensorType2 := FuTypPushbuttonSensorType2(
				bAddress := daliSensors[i].AddrButtons - 1,
				bModule_753_647 := 1
			),
		);
		DaliSensorsInputs[iDali * 12] := DaliButtonT2[i].xButton1;
		DaliSensorsInputs[iDali * 12 + 1] := DaliButtonT2[i].xButton2;
		DaliSensorsInputs[iDali * 12 + 2] := DaliButtonT2[i].xButton3;
		DaliSensorsInputs[iDali * 12 + 3] := DaliButtonT2[i].xButton4;
		DaliSendSensor(i := iDali * 12);
		DaliSendSensor(i := iDali * 12 + 1);
		DaliSendSensor(i := iDali * 12 + 2);
		DaliSendSensor(i := iDali * 12 + 3);

	ELSIF daliSensors[i].SensorType = DaliEcg THEN
		DaliSendValue647[daliSensors[i].Address](
			typBallast := FuTypBallast (
				bAddress :=  daliSensors[i].Address - 1,
				xIsGroup := FALSE,
				bModule_753_647 := 1
			),
			rDimmValue := BYTE_TO_REAL(DaliValue647[daliSensors[i].Address]),
			rHysteresis := 1,
			xUpdate := TRUE
		);
	ELSIF daliSensors[i].SensorType = DaliGroup THEN
		DaliSendValueGrp647[daliSensors[i].Address](
			typBallast := FuTypBallast (
				bAddress :=  daliSensors[i].Address - 1,
				xIsGroup := TRUE,
				bModule_753_647 := 1
			),
			rDimmValue := BYTE_TO_REAL(DaliValueGrp647[daliSensors[i].Address]),
			rHysteresis := 1,
			xUpdate := TRUE
		);

	ELSIF daliSensors[i].SensorType = NoSensor THEN
		(* stop after all devices are processed *)
		EXIT;
	END_IF
END_FOR
END_PROGRAM

(* POU DALI/DaliReadCsvFile, ST *)
PROGRAM DaliReadCsvFile
(*
	This program reads the configuration file for sensors on the DALI multi master bus
	It helps maps the devices to calaos addresses.

	The file calaos_dali_master.csv is read from internal memory
*)
VAR CONSTANT
	sFilename: STRING := 'calaos_dali_master.csv';
	RawDataSize: UINT := 4096;
END_VAR
VAR_IN_OUT
	xStart:	BOOL;
	daliSensors: ARRAY [1..MaxDaliSensors] OF typDaliSensorData;
END_VAR
VAR
	bSeperator:	BYTE := 59; (* seperator semicolon : 59 *)
	bEndLine:	BYTE := 13; (* seperator semicolon : 13 *)
	fd: DWORD;
	rawData: ARRAY[0..RawDataSize] OF BYTE;
	fSize: DWORD;
	tmpStr: STRING;
	startposition: INT;
	i: INT;
	j: INT;
	k: INT;
	paramCount: BYTE;
END_VAR
IF xStart THEN
	fd := SysFileOpen(FileName := sFilename, Mode := 'r');
	IF fd<>0 THEN
		SysFileRead(File:=fd, Buffer:=ADR(rawData), Size:=SIZEOF(rawData));
		fSize:=SysFileGetSize(FileName:=sFilename);
		IF fSize>RawDataSize THEN
			fSize:=RawDataSize;
		END_IF
		SysFileClose(File:=fd);(*this function is blocking*)
	ELSE
		xStart:=FALSE;
		RETURN;(*no such file available*)
	END_IF
(*copy data to typData array*)
	startposition:=0;
	i:=0;
	FOR j:=1 TO MaxDaliSensors DO

		WHILE rawData[startposition+i]<>bSeperator AND
				startposition+i < RawDataSize AND (* File Too  big *)
				rawData[startposition+i] <> 0 DO (* EOF *)
			i:=i+1;
		END_WHILE
		rawData[startposition+i]:=0;
		MEMCPY(pSourceAddress:=ADR(rawData[startposition]), pDestinationAddress:=ADR(tmpStr), BytesToCopy:=i+1);

		IF STRING_COMPARE(tmpStr, 'MultiSensorType1') = TRUE THEN
			daliSensors[j].SensorType := MultiSensorType1;
			daliSensors[j].offDelay := t#10m;
			paramCount := 4;
		ELSIF STRING_COMPARE(tmpStr, 'MultiSensorType2') = TRUE THEN
			daliSensors[j].SensorType := MultiSensorType2;
			daliSensors[j].offDelay := t#10m;
			paramCount := 5;
		ELSIF STRING_COMPARE(tmpStr, 'PushbuttonSensorType1') = TRUE THEN
			daliSensors[j].SensorType := PushbuttonSensorType1;
			paramCount := 5;
		ELSIF STRING_COMPARE(tmpStr, 'PushbuttonSensorType2') = TRUE THEN
			daliSensors[j].SensorType := PushbuttonSensorType2;
			paramCount := 2;
		ELSIF STRING_COMPARE(tmpStr, 'DaliEcg') = TRUE THEN
			daliSensors[j].SensorType := DaliEcg;
			paramCount := 2;
		ELSIF STRING_COMPARE(tmpStr, 'DaliGroup') = TRUE THEN
			daliSensors[j].SensorType := DaliGroup;
			paramCount := 2;
		END_IF

		startposition:=startposition+i+1;
		i:=0;

		(*The parameter values are of type word. The following values are seperated by bSeperator*)
		FOR k:=1 TO paramCount-1 DO
			WHILE rawData[startposition+i]<>bSeperator AND
					rawData[startposition+i]<>bEndLine AND
					rawData[startposition+i]<>0 AND
					startposition+i < RawDataSize DO
				i:=i+1;
			END_WHILE
			rawData[startposition+i]:=0;
			MEMCPY(pSourceAddress:=ADR(rawData[startposition]), pDestinationAddress:=ADR(tmpStr), BytesToCopy:=i+1);

			IF daliSensors[j].SensorType = MultiSensorType1 THEN
				IF k = 1 THEN
					daliSensors[j].AddrPresence := STRING_TO_BYTE(tmpStr);
				ELSIF k = 2 THEN
					daliSensors[j].AddrLightLevel := STRING_TO_BYTE(tmpStr);
				ELSIF k = 3 THEN
					daliSensors[j].offDelay := DWORD_TO_TIME(STRING_TO_DWORD(tmpStr));
				END_IF
			ELSIF daliSensors[j].SensorType = MultiSensorType2 THEN
				IF k = 1 THEN
					daliSensors[j].AddrPresence := STRING_TO_BYTE(tmpStr);
				ELSIF k = 2 THEN
					daliSensors[j].AddrLightLevel := STRING_TO_BYTE(tmpStr);
				ELSIF k = 3 THEN
					daliSensors[j].AddrRemote := STRING_TO_BYTE(tmpStr);
				ELSIF k = 4 THEN
					daliSensors[j].offDelay := DWORD_TO_TIME(STRING_TO_DWORD(tmpStr));
				END_IF
			ELSIF daliSensors[j].SensorType = PushbuttonSensorType1 THEN
				IF k = 1 THEN
					daliSensors[j].AddrButton1 := STRING_TO_BYTE(tmpStr);
				ELSIF k = 2 THEN
					daliSensors[j].AddrButton2 := STRING_TO_BYTE(tmpStr);
				ELSIF k = 3 THEN
					daliSensors[j].AddrButton3 := STRING_TO_BYTE(tmpStr);
				ELSIF k = 4 THEN
					daliSensors[j].AddrButton4 := STRING_TO_BYTE(tmpStr);
				END_IF
			ELSIF daliSensors[j].SensorType = PushbuttonSensorType2 THEN
				IF k = 1 THEN
					daliSensors[j].AddrButtons := STRING_TO_BYTE(tmpStr);
				END_IF
			ELSIF daliSensors[j].SensorType = DaliEcg THEN
				IF k = 1 THEN
					daliSensors[j].Address := STRING_TO_BYTE(tmpStr);
				END_IF
			ELSIF daliSensors[j].SensorType = DaliGroup THEN
				IF k = 1 THEN
					daliSensors[j].Address := STRING_TO_BYTE(tmpStr);
				END_IF
			END_IF

			startposition:=startposition+i;

			IF k = paramCount - 1 THEN
				startposition := startposition + 2;
			ELSE
				startposition := startposition + 1;
			END_IF

			i:=0;
		END_FOR
	END_FOR
(*copy data to array finished*)
	xStart:=FALSE;
END_IF
END_PROGRAM

(* POU MEMCPY, ST *)
(*---------------------------------------------------------------------------------------
  WAGO Kontakttechnik GmbH Hansastr. 27 32423 Minden(Westf.) 
  Tel. +49571/887-0 Fax. +49571/887-0                
                                                                                                
  Project: IEC1131 internal library
  
  Function: MEMCPY
  Description: This function copies BytesToCopy bytes from the source
                         address pSourceAddress to the destination address
                         pDestinationAddress
  Date: 25.09.2000

------------------------------------------------------------------------------------------*)
FUNCTION MEMCPY:BOOL
VAR_INPUT
	pSourceAddress:							POINTER TO ARRAY[1..2] OF BYTE;
	pDestinationAddress:						POINTER TO ARRAY[1..2] OF BYTE;
	BytesToCopy:								DINT;
END_VAR
VAR
END_VAR
WHILE (BytesToCopy > 0) DO
	pDestinationAddress^[1]:=pSourceAddress^[1]; (* copy bytes from source to destination *)
	pDestinationAddress:=ADR(pDestinationAddress^[2]); (* increment destination *)
	pSourceAddress:=ADR(pSourceAddress^[2]);(* increment source *)
	BytesToCopy:=BytesToCopy -1; (* decrement number of bytes to copy *)
END_WHILE
END_FUNCTION

(* POU DALI/DaliSendSensor, ST *)
PROGRAM DaliSendSensor
VAR_INPUT
	i: INT;
END_VAR
VAR
	wBuffer: POINTER TO BYTE;
	command: STRING(255);
	Write: ETHERNET_WRITE_PT;
END_VAR
(* Send a Dali sensor input to calaos_server *)

event[i + 512](IN := DaliSensorsInputs[i]);

IF (event[i + 512].ON = TRUE) THEN
	netDaliSensor[i / 8] := BIT_LOAD_B(netDaliSensor[i / 8], TRUE, i MOD 8);
	command := 'WAGO INT ';
	command := CONCAT(command,  INT_TO_STRING(i + 6656));
	command := CONCAT(command,  ' 1');
	wBuffer := ADR(command);

	Write(EN := 0, SOCKET := 0, LEN_IN := 0, DST_IP:=0, DST_PORT:=0, DATA_PT := wBuffer);
	Write(EN := 1, SOCKET := SendInput.socket, LEN_IN := LEN(command), DST_IP := Config.SERVER_IP, DST_PORT := 4646, DATA_PT := wBuffer);
END_IF
IF (event[i + 512].OFF = TRUE) THEN
	netDaliSensor[i / 8] := BIT_LOAD_B(netDaliSensor[i / 8], FALSE, i MOD 8);
	command := 'WAGO INT ';
	command := CONCAT(command,  INT_TO_STRING(i + 6656));
	command := CONCAT(command,  ' 0');
	wBuffer := ADR(command);

	Write(EN := 0, SOCKET := 0, LEN_IN := 0, DST_IP:=0, DST_PORT:=0, DATA_PT := wBuffer);
	Write(EN := 1, SOCKET := SendInput.socket, LEN_IN := LEN(command), DST_IP := Config.SERVER_IP, DST_PORT := 4646, DATA_PT := wBuffer);
END_IF
END_PROGRAM

(* POU Logic/gate logic/BIT_LOAD_B, ST *)
FUNCTION BIT_LOAD_B : BYTE
VAR_INPUT
	IN : BYTE;
	VAL : BOOL;
	POS : INT;
END_VAR
VAR CONSTANT
	dat : BYTE := 1;
END_VAR

(*
version 1.1	16. mar 2008
programmer 	hugo
tested by	tobias

this function loads a bit into a byte at position pos.
 *)
IF VAL THEN
	BIT_LOAD_B := in OR SHL(dat,pos);
ELSE
	BIT_LOAD_B := in AND (NOT SHL(dat,pos));
END_IF;


(* revision history
hm	29. feb 2008	rev 1.0
	original version

hm	16. mar 2008	rev 1.1
	change input bit to val for compatibility reasons
*)
END_FUNCTION

(* POU Logic/gate logic/BIT_LOAD_DW, ST *)
FUNCTION BIT_LOAD_DW : DWORD
VAR_INPUT
	IN : DWORD;
	VAL : BOOL;
	POS : INT;
END_VAR
VAR CONSTANT
	dat : DWORD := 1;
END_VAR

(*
version 1.1	16. mar 2008
programmer 	hugo
tested by	tobias

this function loads a bit into a DWord at position pos.
 *)
IF val THEN
	BIT_LOAD_DW := in OR SHL(dat,pos);
ELSE
	BIT_LOAD_DW := in AND (NOT SHL(dat,pos));
END_IF;


(* revision history
hm	29. feb 2008	rev 1.0
	original version

hm	16. mar 2008	rev 1.1
	change input bit to val for compatibility reasons
*)
END_FUNCTION

(* POU Logic/gate logic/BIT_LOAD_W, ST *)
FUNCTION BIT_LOAD_W : WORD
VAR_INPUT
	IN : WORD;
	VAL : BOOL;
	POS : INT;
END_VAR
VAR CONSTANT
	dat : WORD := 1;
END_VAR

(*
version 1.1	16. mar 2008
programmer 	hugo
tested by	tobias

this function loads a bit into a Word at position pos.
 *)
IF val THEN
	BIT_LOAD_W := in OR SHL(dat,pos);
ELSE
	BIT_LOAD_W := in AND (NOT SHL(dat,pos));
END_IF;


(* revision history
hm	29. feb 2008	rev 1.0
	original version

hm	16. mar 2008	rev 1.1
	change input bit to val for compatibility reasons
*)
END_FUNCTION

(* POU Logic/gate logic/BYTE_OF_DWORD, ST *)
FUNCTION BYTE_OF_DWORD : BYTE
VAR_INPUT
	in : DWORD;
	N : BYTE;
END_VAR


(*
version 1.2	30. oct. 2008
programmer 	hugo
tested by	oscat

this function extracts a single byte from the nth position from right (right is lowest byte) 
the lower byte (starting with Bit0 from in) is selected with N=0.
*)
BYTE_OF_DWORD := DWORD_TO_BYTE(SHR(in,SHL(n,3)));

(* revision history
hm	17. jan 2007	rev 1.0
	original version

hm	2. jan 2008		rev 1.1
	improved performance

hm	30. oct. 2008	rev 1.2
	improved performance
*)
END_FUNCTION

(* POU Logic/gate logic/BYTE_OF_WORD, ST *)
FUNCTION BYTE_OF_WORD : BYTE
VAR_INPUT
	in : WORD;
	N : BYTE;
END_VAR
BYTE_OF_WORD := WORD_TO_BYTE(SHR(in,n));
END_FUNCTION

(* POU DALI/DaliDimValue, ST *)
FUNCTION_BLOCK DaliDimValue
VAR_INPUT
	xEnable: BOOL := TRUE;
	bShortAddress: BYTE;
	tCycleTime: TIME := t#10s;
	bModule_750_641: BYTE := 1;
END_VAR
VAR_OUTPUT
	xReady: BOOL := TRUE;
	bFeedback: BYTE;
	xStatus: BOOL;
	bDimmValue: BYTE;
END_VAR
VAR
	DimValue641: FbDALI_StatusDimmValue;
	DimValue647: FbDaliShowActualValue;

	axShortAddress: ARRAY [0..63] OF BOOL;
	arActualValue: ARRAY [0..96] OF REAL;
END_VAR
(* Query dim value from an ECG *)

IF Config.CONFIG_DALI = TRUE THEN
	DimValue641(
		xEnable := xEnable,
		bShortAddress := bShortAddress,
		tCycleTime := tCycleTime,
		bModule_750_641 := bModule_750_641,

		xReady => xReady,
		bFeedback => bFeedback,
		xStatus => xStatus,
		bDimmValue => bDimmValue
	);
ELSIF Config.CONFIG_DALI_647 = TRUE THEN
	DimValue647(bModule_753_647 := bModule_750_641);

	bDimmValue := REAL_TO_BYTE(DimValue647.arActualValue[bShortAddress - 1]);
	bFeedback := DimValue647.bFeedback;
END_IF
END_FUNCTION_BLOCK

(* POU DALI/DaliSwitch, ST *)
FUNCTION_BLOCK DaliSwitch
VAR_INPUT
	bAddress: BYTE;
	xGroup: BOOL := FALSE;
	xButton: BOOL;
	bDimmLevel: BYTE;
	bFadeTime: BYTE;
END_VAR
VAR_OUTPUT
END_VAR
VAR
	DaliSendValue641: FbDALI_SwitchValue;
END_VAR
(* A DaliSwitch FB that uses either the 750-641 or 753-647
 Both modules cannot be used at the same time
*)

IF Config.CONFIG_DALI = TRUE THEN
	DaliSendValue641(
		bAddress :=  bAddress,
	    xGroup := xGroup,
		bDimmLevel := bDimmLevel,
		xButton := xButton
	);
ELSIF Config.CONFIG_DALI_647 = TRUE THEN

	IF xGroup = TRUE THEN
		DaliValueGrp647[bAddress] := bDimmLevel;
		IF xButton = FALSE THEN
			DaliSendValueGrp647[bAddress](xUpdate := FALSE);
		END_IF
	ELSE
		DaliValue647[bAddress] := bDimmLevel;
		IF xButton = FALSE THEN
			DaliSendValue647[bAddress](xUpdate := FALSE);
		END_IF
	END_IF

END_IF
END_FUNCTION_BLOCK

(* POU INTER_EVENT, ST *)
FUNCTION_BLOCK INTER_EVENT
VAR_INPUT
	IN: BOOL;
END_VAR
VAR_OUTPUT
	ON: BOOL;
	OFF: BOOL;
END_VAR
VAR
	MTRIG: R_TRIG;
	DTRIG: F_TRIG;
END_VAR
(* Get the ON or OFF event on an input *)

MTRIG(CLK := IN);
ON := MTRIG.Q;
DTRIG(CLK := IN);
OFF := DTRIG.Q;
END_FUNCTION_BLOCK

(* Visualisation DALI 647/DALI_647_Main
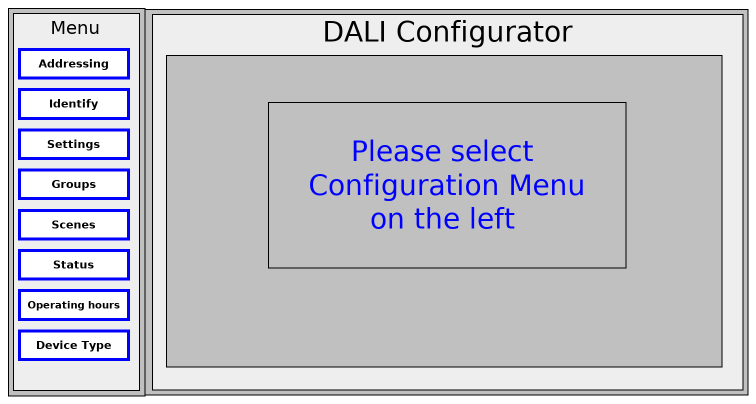
rectangle at (144,6)-(735,382): text "DALI Configurator"
embedded screen at (0,0)-(137,388): visuDALI_Menue
rectangle at (260,94)-(618,260): text "Please select / Configuration Menu / on the left"
2 more shapes without text or variables
*)

(* Visualisation Private/English/visuAddressing
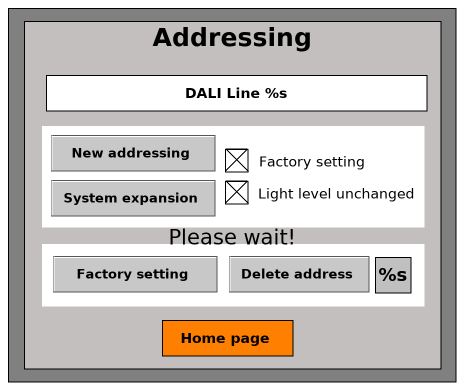
rectangle at (193,71)-(610,419): text "Addressing"
button at (220,185)-(384,221): text "New addressing"; taps DALI_Config.NewAddress; tooltip You have to click and hold the button "New Addressing" longer than two seconds to start the new addressing.
button at (220,230)-(384,266): text "System expansion"; taps DALI_Config.xErweitert; tooltip If you click the button "System expansion", only the ECGs with no short address will be addressed.
rectangle at (544,307)-(580,343): text "%s"; shows DALI_Config.LoeschKurzadr; tooltip Enter the short address to be deleted (1 - 64).; editable
rounded rectangle at (331,370)-(462,406): text "Home page"; opens visuFrontPageDALI; tooltip Back to home page
button at (222,306)-(386,342): text "Factory setting"; taps DALI_Config.Reset; tooltip To reset the ECG you have to click and hold the button two seconds. Group and scene configurations will be deleted.
button at (398,306)-(538,342): text "Delete address"; taps DALI_Config.Loeschen; tooltip The selected short address will be deleted.
rounded rectangle at (215,125)-(596,161): text "DALI Line %s"; shows DALI_Config.Dali_Linie; alarm colour if DALI_Config.keineJobliste; tooltip You can change the DALI Line only on the home page.
rectangle at (426,190)-(537,233): text "Factory setting"
rectangle at (394,231)-(417,254): toggles DALI_Config.xLightLevelUnchanged; tooltip During the addressing, the arc power level will be unchanged. This is only possible, when "Factory setting" is deactivated.
rectangle at (425,221)-(581,266): text "Light level unchanged"
rectangle at (394,199)-(417,222): toggles DALI_Config.FactorySetting; tooltip During the addressing, the control gears will be set to factory default.
polyline at (395,231)-(417,253): invisible if NOT DALI_Config.xLightLevelUnchanged; toggles DALI_Config.xLightLevelUnchanged
polyline at (395,199)-(417,221): invisible if NOT DALI_Config.FactorySetting; toggles DALI_Config.FactorySetting
rectangle at (206,160)-(597,414): text "Please wait!"; invisible if not DALI_Config.JobMerker[5]
3 more shapes without text or variables
*)

(* Visualisation DALI 647/Private/visuDALI_DeviceType_Menue
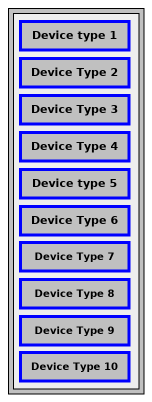
rounded rectangle at (11,49)-(122,80): text "Device Type 2"; alarm colour if dwDeviceType.2; opens DALI_647_DeviceType2_Main; tooltip Discharge lamps,excluding fluorescent lamps.
rounded rectangle at (11,12)-(122,43): text "Device type 1"; alarm colour if dwDeviceType.1; opens DALI_647_DeviceType1_Main; tooltip Self-contained emergency lighting.
rounded rectangle at (11,86)-(122,117): text "Device Type 3"; alarm colour if dwDeviceType.3; opens DALI_647_DeviceType3_Main; tooltip Low voltage halogen lamps
rounded rectangle at (11,123)-(122,154): text "Device Type 4"; alarm colour if dwDeviceType.4; opens DALI_647_DeviceType4_Main; tooltip Supply Voltage controller for incandescent lamps
rounded rectangle at (11,160)-(122,191): text "Device type 5"; alarm colour if dwDeviceType.5; opens DALI_647_DeviceType5_Main; tooltip Conversion from digital into D.C. voltage
rounded rectangle at (11,197)-(122,228): text "Device Type 6"; alarm colour if dwDeviceType.6; opens DALI_647_DeviceType6_Main; tooltip LED modules
rounded rectangle at (11,233)-(122,264): text "Device Type 7"; alarm colour if dwDeviceType.7; opens DALI_647_DeviceType7_Main; tooltip Switching function
rounded rectangle at (11,270)-(122,301): text "Device Type 8"; alarm colour if dwDeviceType.8; opens DALI_647_DeviceType8_Main; tooltip Colour control
rounded rectangle at (11,307)-(122,338): text "Device Type 9"; alarm colour if dwDeviceType.9; opens DALI_647_DeviceType9_Main; tooltip Sequencer
rounded rectangle at (11,343)-(122,374): text "Device Type 10"; alarm colour if dwDeviceType.10; opens DALI_647_DeviceType10_Main; tooltip Optical control
2 more shapes without text or variables
*)

(* Visualisation DALI 647/Private/visuDALI_Menue
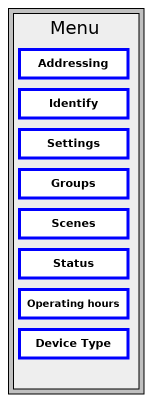
rounded rectangle at (10,80)-(121,111): text "Identify"; opens visuDALIControlGearIdentify
rounded rectangle at (10,40)-(121,71): text "Addressing"; opens visuDALIControlGearAddressing
rounded rectangle at (10,120)-(121,151): text "Settings"; opens visuDALIControlGearSettings
rounded rectangle at (10,160)-(121,191): text "Groups"; opens visuDALIGroups
rounded rectangle at (10,200)-(121,231): text "Scenes"; opens visuDALIScenes
rounded rectangle at (10,240)-(121,271): text "Status"; opens visuDALIControlGearStatus
rounded rectangle at (10,280)-(121,311): text "Operating hours"; opens visuDALIOperatingHours
rounded rectangle at (10,320)-(121,351): text "Device Type"; opens visuDALIDeviceType; tooltip Configuration for other device type
rectangle at (4,8)-(130,38): text "Menu"; opens DALI_647_Main; tooltip Main Page
2 more shapes without text or variables
*)

(* Visualisation DALI 647/Configuration Pages/visuDALIControlGearAddressing
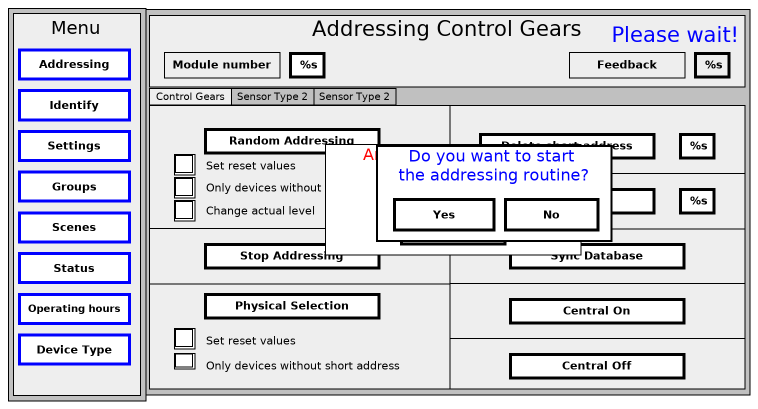
rectangle at (140,7)-(736,79): text "Addressing Control Gears"
rounded rectangle at (155,44)-(271,70): text "Module number"
rounded rectangle at (280,44)-(316,70): text "%s"; shows PrgDALIConfig.bModule_753_647; editable
rounded rectangle at (195,120)-(371,146): text "Random Addressing"; taps PrgDALIConfig.AddressingControlGears.xRandomAddressing
rounded rectangle at (195,285)-(371,311): text "Physical Selection"; taps PrgDALIConfig.AddressingControlGears.xPhysicalSelection
rounded rectangle at (670,125)-(706,151): text "%s"; shows PrgDALIConfig.AddressingControlGears.bDeleteShortAddress; editable 0..63
rounded rectangle at (560,44)-(676,70): text "Feedback"
rounded rectangle at (685,44)-(721,70): text "%s"; shows PrgDALIConfig.AddressingControlGears.bFeedback
rounded rectangle at (500,290)-(676,316): text "Central On"; alarm colour if PrgDALIConfig.AddressingControlGears.xCentralOn; taps PrgDALIConfig.AddressingControlGears.xCentralOn
rounded rectangle at (500,345)-(676,371): text "Central Off"; alarm colour if PrgDALIConfig.AddressingControlGears.xCentralOff; taps PrgDALIConfig.AddressingControlGears.xCentralOff
rectangle at (304,80)-(387,97): text "Sensor Type 2"; invisible if (dwdevicetype.14=FALSE AND dwdevicetype.15=FALSE) OR (dwdevicetype.14=FALSE AND dwdevicetype.15) OR (dwdevicetype.14 AND dwdevicetype.15=FALSE); opens visuDALISensorType2Addressing
rectangle at (140,80)-(223,97): text "Control Gears"
rectangle at (222,80)-(305,97): text "Sensor Type 1"; invisible if (dwdevicetype.14 AND dwdevicetype.15=FALSE) OR (dwdevicetype.14=FALSE AND dwdevicetype.15=FALSE); opens visuDALISensorType1Addressing
rectangle at (222,80)-(305,97): text "Sensor Type 2"; invisible if (dwdevicetype.14=FALSE AND dwdevicetype.15) OR (dwdevicetype.14=FALSE AND dwdevicetype.15=FALSE) OR (dwdevicetype.14 AND dwdevicetype.15); opens visuDALISensorType2Addressing
embedded screen at (165,146)-(186,167): visuDaliSelect
rectangle at (195,145)-(306,171): text "Set reset values"
embedded screen at (165,169)-(186,190): visuDaliSelect
rectangle at (195,167)-(406,193): text "Only devices without short address"
embedded screen at (165,192)-(186,213): visuDaliSelect
rectangle at (195,190)-(336,216): text "Change actual level"
embedded screen at (165,320)-(186,341): visuDaliSelect
rectangle at (195,320)-(306,346): text "Set reset values"
embedded screen at (165,345)-(186,361): visuDaliSelect
rectangle at (195,345)-(406,371): text "Only devices without short address"
rounded rectangle at (470,125)-(646,151): text "Delete short address"; alarm colour if PrgDALIConfig.AddressingControlGears.xDeleteShortAddress; taps PrgDALIConfig.AddressingControlGears.xDeleteShortAddress
rounded rectangle at (670,180)-(706,206): text "%s"; shows PrgDALIConfig.AddressingControlGears.bResetValues; editable
rounded rectangle at (470,180)-(646,206): text "Reset values"; alarm colour if PrgDALIConfig.AddressingControlGears.xResetValues; taps PrgDALIConfig.AddressingControlGears.xResetValues
rounded rectangle at (500,235)-(676,261): text "Sync Database"; alarm colour if PrgDALIConfig.AddressingControlGears.xSyncDataBase; taps PrgDALIConfig.AddressingControlGears.xSyncDataBase
rectangle at (1,13)-(732,382): text "Please wait!"; invisible if PrgDALIConfig.AddressingControlGears.xReady
rounded rectangle at (195,235)-(371,261): text "Stop Addressing"; alarm colour if PrgDALIConfig.AddressingControlGears.xStopAddressing; taps PrgDALIConfig.AddressingControlGears.xStopAddressing
group at (316,136)-(572,247)
  rectangle at (0,0)-(256,111): text "An error has occurred. / Please confirm!"
  rounded rectangle at (75,70)-(181,101): text "Quit"; taps PrgDALIConfig.AddressingControlGears.xQuit
embedded screen at (-1,0)-(137,393): visuDALI_Menue
group at (2,10)-(733,377)
  rectangle at (365,120)-(601,211): text "Do you want to start / the addressing routine?"
  rounded rectangle at (493,170)-(588,201): text "No"; taps PrgDALIConfig.AddressingControlGears.xCancelAddressing
  rounded rectangle at (382,170)-(484,201): text "Yes"; taps PrgDALIConfig.AddressingControlGears.xStartAddressing
10 more shapes without text or variables
*)

(* Visualisation DALI 647/Configuration Pages/visuDALIControlGearIdentify
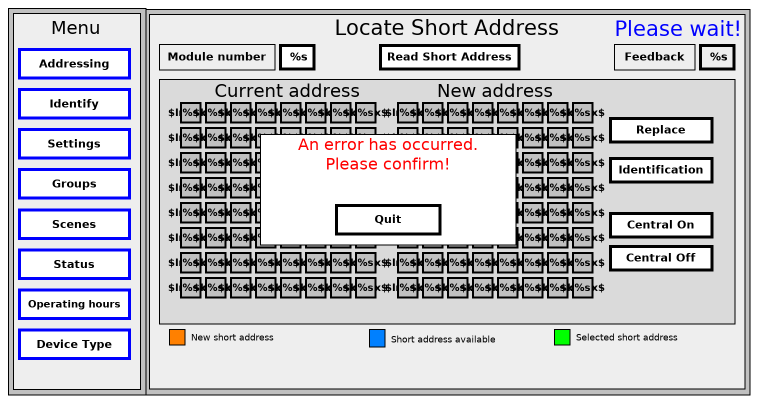
rectangle at (141,6)-(737,381): text "Locate Short Address"
rectangle at (151,71)-(727,316): text "Current address              New address"
rounded rectangle at (151,36)-(267,62): text "Module number"
rounded rectangle at (271,36)-(307,62): text "%s"; shows PrgDALIConfig.bModule_753_647; editable
rectangle at (566,319)-(696,340): text "Selected short address"
rectangle at (381,321)-(502,342): text "Short address available"
rounded rectangle at (606,36)-(687,62): text "Feedback"
rounded rectangle at (691,36)-(727,62): text "%s"; shows PrgDALIConfig.IdentifyControlGear.bFeedback
rounded rectangle at (371,36)-(512,62): text "Read Short Address"; alarm colour if PrgDALIConfig.IdentifyControlGear.xQueryShortAddress; taps PrgDALIConfig.GroupConfig.xQueryShortAddress
rectangle at (181,319)-(311,340): text "New short address"
embedded screen at (0,0)-(138,387): visuDALI_Menue
rounded rectangle at (601,109)-(705,135): text "Replace"; alarm colour if PrgDALIConfig.IdentifyControlGear.xReplaceShortAddress; taps PrgDALIConfig.IdentifyControlGear.xReplaceShortAddress
rounded rectangle at (601,237)-(705,263): text "Central Off"; alarm colour if PrgDALIConfig.IdentifyControlGear.xCentralOff; taps PrgDALIConfig.IdentifyControlGear.xCentralOff
rounded rectangle at (601,204)-(705,230): text "Central On"; alarm colour if PrgDALIConfig.IdentifyControlGear.xCentralOn; taps PrgDALIConfig.IdentifyControlGear.xCentralOn
rounded rectangle at (601,149)-(705,175): text "Identification"; alarm colour if PrgDALIConfig.IdentifyControlGear.xIdentification; toggles PrgDALIConfig.IdentifyControlGear.xIdentification
embedded screen at (172,94)-(193,115): visuIdentifyCurrentAddress
embedded screen at (197,94)-(218,115): visuIdentifyCurrentAddress
embedded screen at (222,94)-(243,115): visuIdentifyCurrentAddress
embedded screen at (247,94)-(268,115): visuIdentifyCurrentAddress
embedded screen at (272,94)-(293,115): visuIdentifyCurrentAddress
embedded screen at (297,94)-(318,115): visuIdentifyCurrentAddress
embedded screen at (322,94)-(343,115): visuIdentifyCurrentAddress
embedded screen at (347,94)-(368,115): visuIdentifyCurrentAddress
embedded screen at (172,119)-(193,140): visuIdentifyCurrentAddress
embedded screen at (197,119)-(218,140): visuIdentifyCurrentAddress
embedded screen at (222,119)-(243,140): visuIdentifyCurrentAddress
embedded screen at (247,119)-(268,140): visuIdentifyCurrentAddress
embedded screen at (272,119)-(293,140): visuIdentifyCurrentAddress
embedded screen at (297,119)-(318,140): visuIdentifyCurrentAddress
embedded screen at (322,119)-(343,140): visuIdentifyCurrentAddress
embedded screen at (347,119)-(368,140): visuIdentifyCurrentAddress
embedded screen at (172,144)-(193,165): visuIdentifyCurrentAddress
embedded screen at (197,144)-(218,165): visuIdentifyCurrentAddress
embedded screen at (222,144)-(243,165): visuIdentifyCurrentAddress
embedded screen at (247,144)-(268,165): visuIdentifyCurrentAddress
embedded screen at (272,144)-(293,165): visuIdentifyCurrentAddress
embedded screen at (297,144)-(318,165): visuIdentifyCurrentAddress
embedded screen at (322,144)-(343,165): visuIdentifyCurrentAddress
embedded screen at (347,144)-(368,165): visuIdentifyCurrentAddress
embedded screen at (172,169)-(193,190): visuIdentifyCurrentAddress
embedded screen at (197,169)-(218,190): visuIdentifyCurrentAddress
embedded screen at (222,169)-(243,190): visuIdentifyCurrentAddress
embedded screen at (247,169)-(268,190): visuIdentifyCurrentAddress
embedded screen at (272,169)-(293,190): visuIdentifyCurrentAddress
embedded screen at (297,169)-(318,190): visuIdentifyCurrentAddress
embedded screen at (322,169)-(343,190): visuIdentifyCurrentAddress
embedded screen at (347,169)-(368,190): visuIdentifyCurrentAddress
embedded screen at (172,194)-(193,215): visuIdentifyCurrentAddress
embedded screen at (197,194)-(218,215): visuIdentifyCurrentAddress
embedded screen at (222,194)-(243,215): visuIdentifyCurrentAddress
embedded screen at (247,194)-(268,215): visuIdentifyCurrentAddress
embedded screen at (272,194)-(293,215): visuIdentifyCurrentAddress
embedded screen at (297,194)-(318,215): visuIdentifyCurrentAddress
embedded screen at (322,194)-(343,215): visuIdentifyCurrentAddress
embedded screen at (347,194)-(368,215): visuIdentifyCurrentAddress
embedded screen at (172,219)-(193,240): visuIdentifyCurrentAddress
embedded screen at (197,219)-(218,240): visuIdentifyCurrentAddress
embedded screen at (222,219)-(243,240): visuIdentifyCurrentAddress
embedded screen at (247,219)-(268,240): visuIdentifyCurrentAddress
embedded screen at (272,219)-(293,240): visuIdentifyCurrentAddress
embedded screen at (297,219)-(318,240): visuIdentifyCurrentAddress
embedded screen at (322,219)-(343,240): visuIdentifyCurrentAddress
embedded screen at (347,219)-(368,240): visuIdentifyCurrentAddress
embedded screen at (172,244)-(193,265): visuIdentifyCurrentAddress
embedded screen at (197,244)-(218,265): visuIdentifyCurrentAddress
embedded screen at (222,244)-(243,265): visuIdentifyCurrentAddress
embedded screen at (247,244)-(268,265): visuIdentifyCurrentAddress
embedded screen at (272,244)-(293,265): visuIdentifyCurrentAddress
embedded screen at (297,244)-(318,265): visuIdentifyCurrentAddress
embedded screen at (322,244)-(343,265): visuIdentifyCurrentAddress
embedded screen at (347,244)-(368,265): visuIdentifyCurrentAddress
embedded screen at (172,269)-(193,290): visuIdentifyCurrentAddress
embedded screen at (197,269)-(218,290): visuIdentifyCurrentAddress
embedded screen at (222,269)-(243,290): visuIdentifyCurrentAddress
embedded screen at (247,269)-(268,290): visuIdentifyCurrentAddress
embedded screen at (272,269)-(293,290): visuIdentifyCurrentAddress
embedded screen at (297,269)-(318,290): visuIdentifyCurrentAddress
embedded screen at (322,269)-(343,290): visuIdentifyCurrentAddress
embedded screen at (347,269)-(368,290): visuIdentifyCurrentAddress
embedded screen at (389,94)-(410,115): visuNewShortAddress
embedded screen at (414,94)-(435,115): visuNewShortAddress
embedded screen at (439,94)-(460,115): visuNewShortAddress
embedded screen at (464,94)-(485,115): visuNewShortAddress
embedded screen at (489,94)-(510,115): visuNewShortAddress
embedded screen at (514,94)-(535,115): visuNewShortAddress
embedded screen at (539,94)-(560,115): visuNewShortAddress
embedded screen at (564,94)-(585,115): visuNewShortAddress
embedded screen at (389,119)-(410,140): visuNewShortAddress
embedded screen at (414,119)-(435,140): visuNewShortAddress
embedded screen at (439,119)-(460,140): visuNewShortAddress
embedded screen at (464,119)-(485,140): visuNewShortAddress
embedded screen at (489,119)-(510,140): visuNewShortAddress
embedded screen at (514,119)-(535,140): visuNewShortAddress
embedded screen at (539,119)-(560,140): visuNewShortAddress
embedded screen at (564,119)-(585,140): visuNewShortAddress
embedded screen at (389,144)-(410,165): visuNewShortAddress
embedded screen at (414,144)-(435,165): visuNewShortAddress
embedded screen at (439,144)-(460,165): visuNewShortAddress
embedded screen at (464,144)-(485,165): visuNewShortAddress
embedded screen at (489,144)-(510,165): visuNewShortAddress
embedded screen at (514,144)-(535,165): visuNewShortAddress
embedded screen at (539,144)-(560,165): visuNewShortAddress
embedded screen at (564,144)-(585,165): visuNewShortAddress
embedded screen at (389,169)-(410,190): visuNewShortAddress
embedded screen at (414,169)-(435,190): visuNewShortAddress
embedded screen at (439,169)-(460,190): visuNewShortAddress
embedded screen at (464,169)-(485,190): visuNewShortAddress
embedded screen at (489,169)-(510,190): visuNewShortAddress
embedded screen at (514,169)-(535,190): visuNewShortAddress
embedded screen at (539,169)-(560,190): visuNewShortAddress
embedded screen at (564,169)-(585,190): visuNewShortAddress
embedded screen at (389,194)-(410,215): visuNewShortAddress
embedded screen at (414,194)-(435,215): visuNewShortAddress
embedded screen at (439,194)-(460,215): visuNewShortAddress
embedded screen at (464,194)-(485,215): visuNewShortAddress
embedded screen at (489,194)-(510,215): visuNewShortAddress
embedded screen at (514,194)-(535,215): visuNewShortAddress
embedded screen at (539,194)-(560,215): visuNewShortAddress
embedded screen at (564,194)-(585,215): visuNewShortAddress
embedded screen at (389,219)-(410,240): visuNewShortAddress
embedded screen at (414,219)-(435,240): visuNewShortAddress
embedded screen at (439,219)-(460,240): visuNewShortAddress
embedded screen at (464,219)-(485,240): visuNewShortAddress
embedded screen at (489,219)-(510,240): visuNewShortAddress
embedded screen at (514,219)-(535,240): visuNewShortAddress
embedded screen at (539,219)-(560,240): visuNewShortAddress
embedded screen at (564,219)-(585,240): visuNewShortAddress
embedded screen at (389,244)-(410,265): visuNewShortAddress
embedded screen at (414,244)-(435,265): visuNewShortAddress
embedded screen at (439,244)-(460,265): visuNewShortAddress
embedded screen at (464,244)-(485,265): visuNewShortAddress
embedded screen at (489,244)-(510,265): visuNewShortAddress
embedded screen at (514,244)-(535,265): visuNewShortAddress
embedded screen at (539,244)-(560,265): visuNewShortAddress
embedded screen at (564,244)-(585,265): visuNewShortAddress
embedded screen at (389,269)-(410,290): visuNewShortAddress
embedded screen at (414,269)-(435,290): visuNewShortAddress
embedded screen at (439,269)-(460,290): visuNewShortAddress
embedded screen at (464,269)-(485,290): visuNewShortAddress
embedded screen at (489,269)-(510,290): visuNewShortAddress
embedded screen at (514,269)-(535,290): visuNewShortAddress
embedded screen at (539,269)-(560,290): visuNewShortAddress
embedded screen at (564,269)-(585,290): visuNewShortAddress
rectangle at (5,7)-(736,378): text "Please wait!"; invisible if PrgDALIConfig.IdentifyControlGear.xReady
group at (252,126)-(508,237)
  rectangle at (0,0)-(256,111): text "An error has occurred. / Please confirm!"
  rounded rectangle at (75,70)-(181,101): text "Quit"; taps PrgDALIConfig.IdentifyControlGear.xQuit
4 more shapes without text or variables
*)

(* Visualisation DALI 647/Configuration Pages/visuDALIControlGearSettings
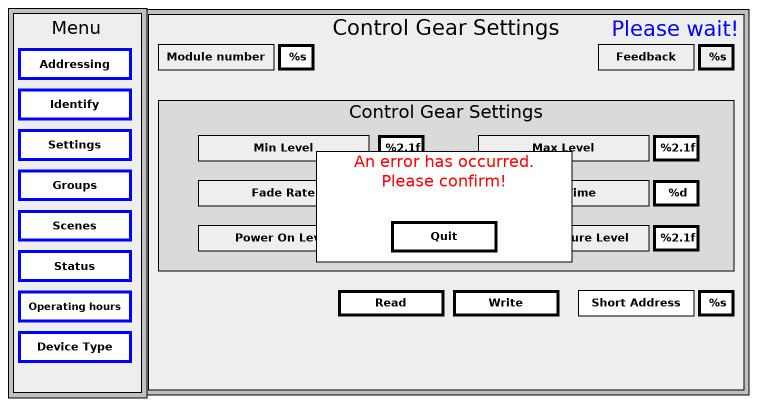
rectangle at (140,6)-(736,382): text "Control Gear Settings"
rounded rectangle at (150,36)-(266,62): text "Module number"
rounded rectangle at (270,36)-(306,62): text "%s"; shows PrgDALIConfig.bModule_753_647; editable
rounded rectangle at (590,36)-(686,62): text "Feedback"
rounded rectangle at (690,36)-(726,62): text "%s"; shows PrgDALIConfig.SettingsControlGear.bFeedback
rounded rectangle at (330,282)-(436,308): text "Read"; alarm colour if PrgDALIConfig.SettingsControlGear.xRead; taps PrgDALIConfig.SettingsControlGear.xRead
rounded rectangle at (445,282)-(551,308): text "Write"; alarm colour if PrgDALIConfig.SettingsControlGear.xWrite; taps PrgDALIConfig.SettingsControlGear.xWrite
rectangle at (150,92)-(726,263): text "Control Gear Settings"
rounded rectangle at (190,127)-(361,153): text "Min Level"
rounded rectangle at (470,127)-(641,153): text "Max Level"
rounded rectangle at (190,172)-(361,198): text "Fade Rate"
rounded rectangle at (470,172)-(641,198): text "Fade Time"
rounded rectangle at (470,217)-(641,243): text "System Failure Level"
rounded rectangle at (190,217)-(361,243): text "Power On Level"
rounded rectangle at (370,127)-(416,153): text "%2.1f"; shows PrgDALIConfig.rMinLevel; editable
rounded rectangle at (370,172)-(416,198): text "%d"; shows PrgDALIConfig.bFadeRate; editable 1..15
rounded rectangle at (370,217)-(416,243): text "%2.1f"; shows PrgDALIConfig.rPowerOnLevel; editable
rounded rectangle at (645,127)-(691,153): text "%2.1f"; shows PrgDALIConfig.rMaxLevel; editable
rounded rectangle at (645,172)-(691,198): text "%d"; shows PrgDALIConfig.bFadeTime; editable 0..15
rounded rectangle at (645,217)-(691,243): text "%2.1f"; shows PrgDALIConfig.rSystemFailureLevel; editable
rounded rectangle at (570,282)-(686,308): text "Group"; invisible if NOT PrgDALIConfig.SettingsControlGear.typBallast.xIsGroup; toggles PrgDALIConfig.SettingsControlGear.typBallast.xIsGroup
rounded rectangle at (570,282)-(686,308): text "Short Address"; invisible if PrgDALIConfig.SettingsControlGear.typBallast.xIsGroup; toggles PrgDALIConfig.SettingsControlGear.typBallast.xIsGroup
rounded rectangle at (690,282)-(726,308): text "%s"; shows PrgDALIConfig.SettingsControlGear.typBallast.bAddress; editable
embedded screen at (0,0)-(139,390): visuDALI_Menue
rectangle at (2,7)-(733,376): text "Please wait!"; invisible if PrgDALIConfig.SettingsControlGear.xReady
group at (308,143)-(564,254)
  rectangle at (0,0)-(256,111): text "An error has occurred. / Please confirm!"
  rounded rectangle at (75,70)-(181,101): text "Quit"; taps PrgDALIConfig.SettingsControlGear.xQuit
1 more shapes without text or variables
*)

(* Visualisation DALI 647/Configuration Pages/visuDALIControlGearStatus
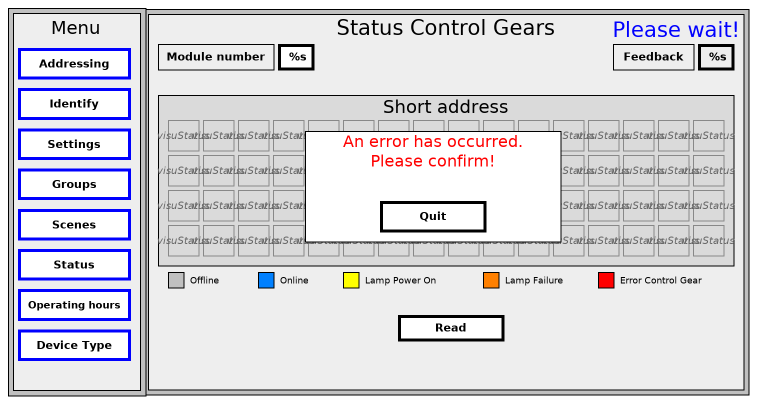
rectangle at (140,6)-(736,382): text "Status Control Gears"
rectangle at (150,87)-(726,258): text "Short address"
embedded screen at (160,112)-(191,143): visuStatus
embedded screen at (195,112)-(226,143): visuStatus
embedded screen at (230,112)-(261,143): visuStatus
embedded screen at (265,112)-(296,143): visuStatus
embedded screen at (300,112)-(331,143): visuStatus
embedded screen at (335,112)-(366,143): visuStatus
embedded screen at (370,112)-(401,143): visuStatus
embedded screen at (405,112)-(436,143): visuStatus
rounded rectangle at (150,36)-(266,62): text "Module number"
rounded rectangle at (270,36)-(306,62): text "%s"; shows PrgDALIConfig.bModule_753_647; editable
rounded rectangle at (605,36)-(686,62): text "Feedback"
rounded rectangle at (690,36)-(726,62): text "%s"; shows PrgDALIConfig.StatusControlGear.bFeedback
embedded screen at (440,112)-(471,143): visuStatus
embedded screen at (475,112)-(506,143): visuStatus
embedded screen at (510,112)-(541,143): visuStatus
embedded screen at (545,112)-(576,143): visuStatus
embedded screen at (580,112)-(611,143): visuStatus
embedded screen at (615,112)-(646,143): visuStatus
embedded screen at (650,112)-(681,143): visuStatus
embedded screen at (685,112)-(716,143): visuStatus
embedded screen at (160,147)-(191,178): visuStatus
embedded screen at (195,147)-(226,178): visuStatus
embedded screen at (230,147)-(261,178): visuStatus
embedded screen at (265,147)-(296,178): visuStatus
embedded screen at (300,147)-(331,178): visuStatus
embedded screen at (335,147)-(366,178): visuStatus
embedded screen at (370,147)-(401,178): visuStatus
embedded screen at (405,147)-(436,178): visuStatus
embedded screen at (440,147)-(471,178): visuStatus
embedded screen at (475,147)-(506,178): visuStatus
embedded screen at (510,147)-(541,178): visuStatus
embedded screen at (545,147)-(576,178): visuStatus
embedded screen at (580,147)-(611,178): visuStatus
embedded screen at (615,147)-(646,178): visuStatus
embedded screen at (650,147)-(681,178): visuStatus
embedded screen at (685,147)-(716,178): visuStatus
embedded screen at (160,182)-(191,213): visuStatus
embedded screen at (195,182)-(226,213): visuStatus
embedded screen at (230,182)-(261,213): visuStatus
embedded screen at (265,182)-(296,213): visuStatus
embedded screen at (300,182)-(331,213): visuStatus
embedded screen at (335,182)-(366,213): visuStatus
embedded screen at (370,182)-(401,213): visuStatus
embedded screen at (405,182)-(436,213): visuStatus
embedded screen at (440,182)-(471,213): visuStatus
embedded screen at (475,182)-(506,213): visuStatus
embedded screen at (510,182)-(541,213): visuStatus
embedded screen at (545,182)-(576,213): visuStatus
embedded screen at (580,182)-(611,213): visuStatus
embedded screen at (615,182)-(646,213): visuStatus
embedded screen at (650,182)-(681,213): visuStatus
embedded screen at (685,182)-(716,213): visuStatus
embedded screen at (160,217)-(191,248): visuStatus
embedded screen at (195,217)-(226,248): visuStatus
embedded screen at (230,217)-(261,248): visuStatus
embedded screen at (265,217)-(296,248): visuStatus
embedded screen at (300,217)-(331,248): visuStatus
embedded screen at (335,217)-(366,248): visuStatus
embedded screen at (370,217)-(401,248): visuStatus
embedded screen at (405,217)-(436,248): visuStatus
embedded screen at (440,217)-(471,248): visuStatus
embedded screen at (475,217)-(506,248): visuStatus
embedded screen at (510,217)-(541,248): visuStatus
embedded screen at (545,217)-(576,248): visuStatus
embedded screen at (580,217)-(611,248): visuStatus
embedded screen at (615,217)-(646,248): visuStatus
embedded screen at (650,217)-(681,248): visuStatus
embedded screen at (685,217)-(716,248): visuStatus
rounded rectangle at (390,307)-(496,333): text "Read"; alarm colour if PrgDALIConfig.StatusControlGear.xRead; taps PrgDALIConfig.StatusControlGear.xRead
rectangle at (270,262)-(371,283): text "Online"
rectangle at (180,262)-(310,283): text "Offline"
rectangle at (495,262)-(591,283): text "Lamp Failure"
rectangle at (355,262)-(451,283): text "Lamp Power On"
rectangle at (610,262)-(706,283): text "Error Control Gear"
embedded screen at (0,0)-(138,388): visuDALI_Menue
rectangle at (3,8)-(734,381): text "Please wait!"; invisible if PrgDALIConfig.StatusControlGear.xReady
group at (297,123)-(553,234)
  rectangle at (0,0)-(256,111): text "An error has occurred. / Please confirm!"
  rounded rectangle at (75,70)-(181,101): text "Quit"; taps PrgDALIConfig.StatusControlGear.xQuit
6 more shapes without text or variables
*)

(* Visualisation DALI 647/Configuration Pages/visuDALIDeviceType
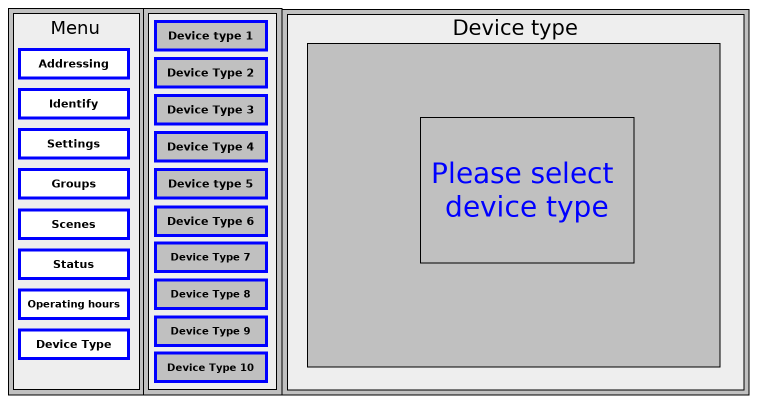
rectangle at (279,6)-(736,382): text "Device type"
embedded screen at (0,0)-(137,387): visuDALI_Menue
embedded screen at (135,0)-(274,387): visuDALI_DeviceType_Menue
rectangle at (412,109)-(626,255): text "Please select / device type"
2 more shapes without text or variables
*)

